CASE eState OF
    CFF_IDLE:
        bBusy := FALSE;
        bDone := FALSE;
        bError := FALSE;
        bAborted := FALSE;
        stFastConfigSnapshot.bValid := FALSE;
        IF bStartEvent THEN
            udiActiveStartCommandId := GVL_FastInternal.stAcceptedCommand.stSequence.nCommandId;
            stActiveSequenceCommand := GVL_FastInternal.stAcceptedCommand.stSequence;
            udiActiveCycleSnapshotRevision := GVL_FastInternal.stAcceptedCommand.nCycleSnapshotRevision;
            udiStartCycleSnapshotRevisionBefore := GVL_Program.stCycleSnapshot.nSnapshotRevision;
            udiStartMachineRevisionBefore := GVL_Config.stMachine.nRevision;
            udiStartForceProfileIdBefore := GVL_Config.stZForceControl.nProfileId;
            udiStartForceProfileRevisionBefore := GVL_Config.stZForceControl.nRevision;
            udiStartRAxisProfileIdBefore := GVL_Config.stRAxis.nProfileId;
            udiStartRAxisProfileRevisionBefore := GVL_Config.stRAxis.nRevision;
            stCycleSnapshot := GVL_Program.stCycleSnapshot;
            stMachineSnapshot := GVL_Config.stMachine;
            stLimitsSnapshot := GVL_Config.stLimits;
            stSequenceConfigSnapshot := GVL_Config.stCffSequence;
            stZExtConfigSnapshot := GVL_Config.stZExtSetpoint;
            stForceProfileSnapshot := GVL_Config.stZForceControl;
            stRAxisProfileSnapshot := GVL_Config.stRAxis;
            bStartSourceSnapshotConsistent :=
                (udiStartCycleSnapshotRevisionBefore = stCycleSnapshot.nSnapshotRevision)
                AND (GVL_Program.stCycleSnapshot.nSnapshotRevision
                    = stCycleSnapshot.nSnapshotRevision)
                AND (udiStartMachineRevisionBefore = stMachineSnapshot.nRevision)
                AND (GVL_Config.stMachine.nRevision = stMachineSnapshot.nRevision)
                AND (udiStartForceProfileIdBefore = stForceProfileSnapshot.nProfileId)
                AND (udiStartForceProfileRevisionBefore = stForceProfileSnapshot.nRevision)
                AND (GVL_Config.stZForceControl.nProfileId = stForceProfileSnapshot.nProfileId)
                AND (GVL_Config.stZForceControl.nRevision = stForceProfileSnapshot.nRevision)
                AND (udiStartRAxisProfileIdBefore = stRAxisProfileSnapshot.nProfileId)
                AND (udiStartRAxisProfileRevisionBefore = stRAxisProfileSnapshot.nRevision)
                AND (GVL_Config.stRAxis.nProfileId = stRAxisProfileSnapshot.nProfileId)
                AND (GVL_Config.stRAxis.nRevision = stRAxisProfileSnapshot.nRevision);
            rCycleStartZPosition_mm := GVL_Status.stFast.stZAxis.rActualPosition_mm;
            bBusy := TRUE;
            bCycleNokLatched := FALSE;
            bStopRequestedLatched := FALSE;
            bResetPendingLatched := FALSE;
            udiFirstFaultId :=0;
            eExitIntent := CFF_EXIT_NONE;
            eStep := CFF_STEP_NONE;
            eSubPhase := STEP_SUBPHASE_NONE;
            eEndCause := STEP_END_NONE;
            FOR nStepIndex := 1 TO 4 DO
                GVL_Process.astStepCriterion[nStepIndex] := stClearedStepCriterionResult;
                abStepResultWritten[nStepIndex] := FALSE;
            END_FOR
            stLastPublishedRCommand.bEnable := TRUE;
            stLastPublishedRCommand.bReset := FALSE;
            stLastPublishedRCommand.bStop := TRUE;
            stLastPublishedRCommand.bMoveVelocity := FALSE;
            stLastPublishedRCommand.rVelocity_rpm := 0.0;
            stLastPublishedRCommand.rAcceleration_rpm_s :=
                stRAxisProfileSnapshot.fSpeedRampRpmS;
            stLastPublishedRCommand.rDeceleration_rpm_s :=
                stRAxisProfileSnapshot.fSpeedRampRpmS;
            stCandidateRCommand := stLastPublishedRCommand;
            rHardMaximumRelativePosition_mm := 0.0;
            rRequiredRelativePosition_mm := 0.0;
            rStepBoundary_mm := 0.0;
            rForceTransferVelocity_mm_s := 0.0;
            rForceSet_kN := 0.0;
            rForceRamp_kN_s := 0.0;
            rSpeedSet_rpm := 0.0;
            rTargetRelativePosition_mm := 0.0;
            rStepTime_s := 0.0;
            rQualifiedForceHoldTime_s := 0.0;
            uliStepElapsed_us := 0;
            uliStepMaximum_us := 0;
            uliQualifiedHold_us := 0;
            uliQualifiedHoldTarget_us := 0;
            bRpmStopped := FALSE;
            bForceInBand := FALSE;
            bHardForceActive := FALSE;
            bHardStrokeActive := FALSE;
            bCollisionLimitActive := FALSE;
            bForceControlEnable := FALSE;
            bForceProfileTransfer := FALSE;
            bForceProfileTransferPending := FALSE;
            bProcessReferencePending := FALSE;
            bProcessReferenceResetPending := FALSE;
            bProcessReferenceLatchPending := FALSE;
            bApproachFaultStopPending := FALSE;
            bUnknownExternalRStopPending := FALSE;
            bSafeExitRStopPending := FALSE;
            bTerminalFaultStopRequired := FALSE;
            bUnloadTransferInitialized := FALSE;
            stFastConfigSnapshot.bValid := FALSE;
            eNextState := CFF_PRECHECK;
        END_IF

    CFF_PRECHECK:
        (* Generate the first of the two local Contact transactions: Reset. *)
        IF bStateEntry THEN
            IF NOT bProcessReferencePending THEN
                stPendingProcessReferenceCommand.bLatchContactReference := FALSE;
                stPendingProcessReferenceCommand.bUseProvidedContactReference := FALSE;
                stPendingProcessReferenceCommand.rProvidedContactSensorPosition_mm := 0.0;
                stPendingProcessReferenceCommand.rProvidedContactAxisPosition_mm := 0.0;
                stPendingProcessReferenceCommand.bResetContactReference := TRUE;
                udiContactReferenceRequestId := udiContactReferenceRequestId + 1;
                IF udiContactReferenceRequestId = 0 THEN
                    udiContactReferenceRequestId := 1;
                END_IF
                stPendingProcessReferenceCommand.udiContactReferenceRequestId := udiContactReferenceRequestId;
                udiExpectedContactReferenceAckId := udiContactReferenceRequestId;
                bProcessReferencePending := TRUE;
                bProcessReferenceResetPending := TRUE;
                bProcessReferenceLatchPending := FALSE;
            END_IF
        END_IF

        IF bProcessReferenceResetPending
            AND (GVL_Process.stActual.udiContactReferenceAcceptedId
                = udiExpectedContactReferenceAckId) THEN
            bProcessReferencePending := FALSE;
            bProcessReferenceResetPending := FALSE;
            IF GVL_Process.stActual.bContactReferenceValid THEN
                IF udiFirstFaultId = 0 THEN
                    udiFirstFaultId := 16#0000A001;
                END_IF
                eNextState := CFF_FAULT;
            ELSIF bPermissionValid AND bSnapshotIdentityValid
                AND stMachineSnapshot.bValid AND stLimitsSnapshot.bValid
                AND stCycleSnapshot.stProgram.bValid AND stZExtConfigSnapshot.bValid
                AND bProgramValid AND bSequenceConfigValid AND bProfileValid
                AND bHardwareReady AND bSensorReady AND bLocalReturnTargetValid
                AND bExternalReady
                AND (GVL_Status.stFast.stZAxis.eActiveOwner = Z_OWNER_NONE) THEN
                stFastConfigSnapshot.nSequenceCommandId := udiActiveStartCommandId;
                stFastConfigSnapshot.stMachine := stMachineSnapshot;
                stFastConfigSnapshot.stLimits := stLimitsSnapshot;
                stFastConfigSnapshot.stZExtSetpoint := stZExtConfigSnapshot;
                stFastConfigSnapshot.stZForceControl := stForceProfileSnapshot;
                stFastConfigSnapshot.bValid := TRUE;
                eNextState := CFF_APPROACH;
            ELSE
                IF udiFirstFaultId = 0 THEN
                    IF NOT bPermissionValid OR NOT bSnapshotIdentityValid THEN
                        udiFirstFaultId := 16#0000A001;
                    ELSIF NOT bProgramValid THEN
                        udiFirstFaultId := 16#0000A002;
                    ELSIF NOT bSequenceConfigValid OR NOT stMachineSnapshot.bValid
                        OR NOT stLimitsSnapshot.bValid OR NOT stZExtConfigSnapshot.bValid THEN
                        udiFirstFaultId := 16#0000A003;
                    ELSIF NOT bProfileValid THEN
                        udiFirstFaultId := 16#0000A004;
                    ELSIF NOT bHardwareReady THEN
                        udiFirstFaultId := 16#0000A005;
                    ELSE
                        udiFirstFaultId := 16#0000A006;
                    END_IF
                END_IF
                stFastConfigSnapshot.bValid := FALSE;
                eExitIntent := CFF_EXIT_FAULT_NO_RETURN;
                eNextState := CFF_FAULT;
            END_IF
        ELSIF tonContactReferenceAck.Q THEN
            IF udiFirstFaultId = 0 THEN
                udiFirstFaultId := 16#0000A009;
            END_IF
            stFastConfigSnapshot.bValid := FALSE;
            eExitIntent := CFF_EXIT_FAULT_NO_RETURN;
            eNextState := CFF_FAULT;
        END_IF

    CFF_APPROACH:
        stMotionIntent.stZCommand.bEnable := TRUE;
        stMotionIntent.stZCommand.bReset := FALSE;
        stMotionIntent.stZCommand.bStop := FALSE;
        stMotionIntent.stZCommand.bHome := FALSE;
        stMotionIntent.stZCommand.bMoveAbsolute := TRUE;
        stMotionIntent.stZCommand.bMoveVelocity := FALSE;
        stMotionIntent.stZCommand.bUseExternalSetpoint := FALSE;
        stMotionIntent.stZCommand.rPosition_mm := stCycleSnapshot.stProgram.stHeader.fContactSearchStartPositionMm;
        stMotionIntent.stZCommand.rVelocity_mm_s := stCycleSnapshot.stProgram.stHeader.fContactSearchVelocityMmS;
        stMotionIntent.stZCommand.rAcceleration_mm_s2 := stSequenceConfigSnapshot.fStandardMoveAccelerationMmS2;
        stMotionIntent.stZCommand.rDeceleration_mm_s2 := stSequenceConfigSnapshot.fStandardMoveDecelerationMmS2;
        stMotionIntent.stZCommand.eOwnerRequest := Z_OWNER_APPROACH;
        stMotionIntent.bRAxisProcessRequested := TRUE;
        stMotionIntent.stRCommand.bEnable := TRUE;
        stMotionIntent.stRCommand.bReset := FALSE;
        stMotionIntent.stRCommand.bStop := TRUE;
        stMotionIntent.stRCommand.bMoveVelocity := FALSE;
        stMotionIntent.stRCommand.rVelocity_rpm := 0.0;
        stMotionIntent.stRCommand.rAcceleration_rpm_s := stRAxisProfileSnapshot.fSpeedRampRpmS;
        stMotionIntent.stRCommand.rDeceleration_rpm_s := stRAxisProfileSnapshot.fSpeedRampRpmS;
        IF bStateEntry THEN
            IF bEntryMotionPermitted THEN
                udiZCommandId := udiZCommandId + 1;
                IF udiZCommandId = 0 THEN
                    udiZCommandId := 1;
                END_IF
            END_IF
            udiRCommandId := udiRCommandId + 1;
            IF udiRCommandId = 0 THEN
                udiRCommandId := 1;
            END_IF
        END_IF
        IF bApproachNormalCompletion THEN
            eNextState := CFF_EXTSETPOINT_PREPARE;
        ELSIF tonRAxisStop.Q THEN
            IF udiFirstFaultId = 0 THEN
                udiFirstFaultId := 16#0000A014;
            END_IF
            eExitIntent := CFF_EXIT_FAULT_NO_RETURN;
            eNextState := CFF_FAULT;
        ELSIF tonApproach.Q THEN
            IF udiFirstFaultId = 0 THEN
                udiFirstFaultId := 16#0000A007;
            END_IF
            eExitIntent := CFF_EXIT_FAULT_NO_RETURN;
            eNextState := CFF_FAULT;
        ELSIF GVL_Status.stFast.stZAxis.bError THEN
            IF udiFirstFaultId = 0 THEN
                udiFirstFaultId := 16#0000A010;
            END_IF
            eExitIntent := CFF_EXIT_FAULT_NO_RETURN;
            eNextState := CFF_FAULT;
        ELSIF GVL_Status.stFast.stRAxis.bError THEN
            IF udiFirstFaultId = 0 THEN
                udiFirstFaultId := 16#0000A011;
            END_IF
            eExitIntent := CFF_EXIT_FAULT_NO_RETURN;
            eNextState := CFF_FAULT;
        END_IF

    CFF_EXTSETPOINT_PREPARE:
        stMotionIntent.stZCommand.bEnable := TRUE;
        stMotionIntent.stZCommand.bUseExternalSetpoint := TRUE;
        stMotionIntent.stZCommand.eOwnerRequest := Z_OWNER_FORCE_PROCESS;
        stMotionIntent.bExternalEnableRequest := TRUE;
        stMotionIntent.bExternalDisableRequest := FALSE;
        stMotionIntent.bRAxisProcessRequested := TRUE;
        stMotionIntent.stRCommand.bEnable := TRUE;
        stMotionIntent.stRCommand.bStop := TRUE;
        stMotionIntent.stRCommand.bMoveVelocity := FALSE;
        stMotionIntent.stRCommand.rVelocity_rpm := 0.0;
        stMotionIntent.stRCommand.rAcceleration_rpm_s := stRAxisProfileSnapshot.fSpeedRampRpmS;
        stMotionIntent.stRCommand.rDeceleration_rpm_s := stRAxisProfileSnapshot.fSpeedRampRpmS;
        bForceControlEnable := FALSE;
        IF bStateEntry THEN
            udiZCommandId := udiZCommandId + 1;
            IF udiZCommandId = 0 THEN
                udiZCommandId := 1;
            END_IF
        END_IF
        IF (GVL_Status.stFast.udiAcceptedSequenceZCommandId = udiZCommandId)
            AND (GVL_Status.stFast.stZAxis.eActiveOwner = Z_OWNER_FORCE_PROCESS)
            AND GVL_Status.stFast.stZExtSetpoint.bEnabled
            AND GVL_Status.stFast.stZExtSetpoint.bAcceptedSetpointValid
            AND GVL_Status.stFast.stZExternalTrajectory.bActive THEN
            eNextState := CFF_CONTACT_SEARCH;
        END_IF

    CFF_CONTACT_SEARCH:
        stMotionIntent.stZCommand.bEnable := TRUE;
        stMotionIntent.stZCommand.bUseExternalSetpoint := TRUE;
        stMotionIntent.stZCommand.eOwnerRequest := Z_OWNER_FORCE_PROCESS;
        stMotionIntent.bExternalEnableRequest := TRUE;
        stMotionIntent.bExternalDisableRequest := FALSE;
        stMotionIntent.rExternalTargetVelocity_mm_s := ABS(stCycleSnapshot.stProgram.stHeader.fContactSearchVelocityMmS);
        stMotionIntent.bRAxisProcessRequested := TRUE;
        stMotionIntent.stRCommand.bEnable := TRUE;
        stMotionIntent.stRCommand.bStop := TRUE;
        stMotionIntent.stRCommand.bMoveVelocity := FALSE;
        stMotionIntent.stRCommand.rVelocity_rpm := 0.0;
        stMotionIntent.stRCommand.rAcceleration_rpm_s := stRAxisProfileSnapshot.fSpeedRampRpmS;
        stMotionIntent.stRCommand.rDeceleration_rpm_s := stRAxisProfileSnapshot.fSpeedRampRpmS;
        bForceControlEnable := FALSE;
        IF fbContactDetect.stOutput.bReferenceLatchRequest AND NOT bProcessReferencePending THEN
            stPendingProcessReferenceCommand.bLatchContactReference := TRUE;
            stPendingProcessReferenceCommand.bUseProvidedContactReference := TRUE;
            stPendingProcessReferenceCommand.rProvidedContactSensorPosition_mm := fbContactDetect.stOutput.rDetectedSensorPosition_mm;
            stPendingProcessReferenceCommand.rProvidedContactAxisPosition_mm := fbContactDetect.stOutput.rDetectedAxisPosition_mm;
            stPendingProcessReferenceCommand.bResetContactReference := FALSE;
            udiContactReferenceRequestId := udiContactReferenceRequestId + 1;
            IF udiContactReferenceRequestId = 0 THEN
                udiContactReferenceRequestId := 1;
            END_IF
            stPendingProcessReferenceCommand.udiContactReferenceRequestId := udiContactReferenceRequestId;
            udiExpectedContactReferenceAckId := udiContactReferenceRequestId;
            bProcessReferencePending := TRUE;
            bProcessReferenceResetPending := FALSE;
            bProcessReferenceLatchPending := TRUE;
            eNextState := CFF_CONTACT_ACCEPT;
        ELSIF tonContactSearch.Q OR fbContactDetect.stOutput.bFault THEN
            IF udiFirstFaultId = 0 THEN
                udiFirstFaultId := 16#0000A008;
            END_IF
            eExitIntent := CFF_EXIT_FAULT_NO_RETURN;
            eNextState := CFF_EXTSETPOINT_DISABLE;
        END_IF

    CFF_CONTACT_ACCEPT:
        stMotionIntent.stZCommand.bEnable := TRUE;
        stMotionIntent.stZCommand.bUseExternalSetpoint := TRUE;
        stMotionIntent.stZCommand.eOwnerRequest := Z_OWNER_FORCE_PROCESS;
        stMotionIntent.bExternalEnableRequest := TRUE;
        stMotionIntent.bExternalDisableRequest := FALSE;
        stMotionIntent.rExternalTargetVelocity_mm_s := ABS(stCycleSnapshot.stProgram.stHeader.fContactSearchVelocityMmS);
        stMotionIntent.bRAxisProcessRequested := TRUE;
        stMotionIntent.stRCommand.bEnable := TRUE;
        stMotionIntent.stRCommand.bStop := TRUE;
        stMotionIntent.stRCommand.bMoveVelocity := FALSE;
        stMotionIntent.stRCommand.rVelocity_rpm := 0.0;
        stMotionIntent.stRCommand.rAcceleration_rpm_s := stRAxisProfileSnapshot.fSpeedRampRpmS;
        stMotionIntent.stRCommand.rDeceleration_rpm_s := stRAxisProfileSnapshot.fSpeedRampRpmS;
        bForceControlEnable := FALSE;
        IF bProcessReferenceLatchPending
            AND (GVL_Process.stActual.udiContactReferenceAcceptedId
                = udiExpectedContactReferenceAckId) THEN
            bProcessReferencePending := FALSE;
            bProcessReferenceLatchPending := FALSE;
            IF NOT GVL_Process.stActual.bContactReferenceValid THEN
                IF udiFirstFaultId = 0 THEN
                    udiFirstFaultId := 16#0000A00A;
                END_IF
                eExitIntent := CFF_EXIT_FAULT_NO_RETURN;
                eNextState := CFF_EXTSETPOINT_DISABLE;
            ELSIF NOT GVL_Process.stActual.bAxisSensorAgreement
                OR NOT GVL_Process.stActual.bValid THEN
                IF udiFirstFaultId = 0 THEN
                    udiFirstFaultId := 16#0000A00F;
                END_IF
                eExitIntent := CFF_EXIT_FAULT_NO_RETURN;
                eNextState := CFF_EXTSETPOINT_DISABLE;
            ELSE
                rHardMaximumRelativePosition_mm := stLimitsSnapshot.fZMaxPositionMm
                    - GVL_Process.stActual.fContactAxisPositionMm;
                rRequiredRelativePosition_mm := 0.0;
                FOR nStepIndex := 1 TO 4 DO
                    rStepBoundary_mm := stCycleSnapshot.stProgram.astSteps[nStepIndex].stProceeding.fRelativeDistanceMm;
                    IF stCycleSnapshot.stProgram.astSteps[nStepIndex].stProceeding.fSecondarySRelMm
                        > rStepBoundary_mm THEN
                        rStepBoundary_mm := stCycleSnapshot.stProgram.astSteps[nStepIndex].stProceeding.fSecondarySRelMm;
                    END_IF
                    IF rStepBoundary_mm > rRequiredRelativePosition_mm THEN
                        rRequiredRelativePosition_mm := rStepBoundary_mm;
                    END_IF
                END_FOR
                IF NOT FC_IsFiniteLReal(rValue := rHardMaximumRelativePosition_mm)
                    OR (rHardMaximumRelativePosition_mm <= 0.0)
                    OR (rRequiredRelativePosition_mm > rHardMaximumRelativePosition_mm) THEN
                    IF udiFirstFaultId = 0 THEN
                        udiFirstFaultId := 16#0000A00D;
                    END_IF
                    eExitIntent := CFF_EXIT_FAULT_NO_RETURN;
                    eNextState := CFF_EXTSETPOINT_DISABLE;
                ELSE
                    rForceTransferVelocity_mm_s := GVL_Status.stFast.stZExtSetpoint.rAcceptedVelocity_mm_s;
                    rForceSet_kN := GVL_Process.stActual.fForceControlN * 0.001;
                    rForceRamp_kN_s := stForceProfileSnapshot.fForceRampNS * 0.001;
                    bForceProfileTransferPending := TRUE;
                    bForceControlEnable := TRUE;
                    eNextState := CFF_STEP1_ENTRY;
                END_IF
            END_IF
        ELSIF tonContactReferenceAck.Q THEN
            IF udiFirstFaultId = 0 THEN
                udiFirstFaultId := 16#0000A009;
            END_IF
            eExitIntent := CFF_EXIT_FAULT_NO_RETURN;
            eNextState := CFF_EXTSETPOINT_DISABLE;
        END_IF

    (* Step1 Entry：同一扫描发布Force目标、R目标和一次事务。 *)
    CFF_STEP1_ENTRY:
        stMotionIntent.stZCommand.bEnable := TRUE;
        stMotionIntent.stZCommand.bUseExternalSetpoint := TRUE;
        stMotionIntent.stZCommand.eOwnerRequest := Z_OWNER_FORCE_PROCESS;
        stMotionIntent.bExternalEnableRequest := TRUE;
        stMotionIntent.bRAxisProcessRequested := TRUE;
        stMotionIntent.stRCommand := stLastPublishedRCommand;
        bForceControlEnable := TRUE;
        eStep := CFF_STEP1_PENETRATION;
        eSubPhase := STEP_SUBPHASE_ENTRY;
        IF bStateEntry AND bEntryMotionPermitted THEN
            rForceSet_kN := stCycleSnapshot.stProgram.astSteps[1].fSetForceN * 0.001;
            rForceRamp_kN_s := stCycleSnapshot.stProgram.astSteps[1].fForceRampNS * 0.001;
            rSpeedSet_rpm := stCycleSnapshot.stProgram.astSteps[1].fSetSpeedRpm;
            IF stCycleSnapshot.stProgram.astSteps[nActiveStepProgramIndex].stProceeding.ePrimaryCriterion
                = STEP_CRIT_RELATIVE_DISTANCE THEN
                rTargetRelativePosition_mm :=
                    stCycleSnapshot.stProgram.astSteps[nActiveStepProgramIndex].stProceeding.fRelativeDistanceMm;
            ELSE
                rTargetRelativePosition_mm :=
                    stCycleSnapshot.stProgram.astSteps[nActiveStepProgramIndex].stProceeding.fSecondarySRelMm;
            END_IF
            rForceTransferVelocity_mm_s :=
                GVL_Status.stFast.stZExtSetpoint.rAcceptedVelocity_mm_s;
            bForceProfileTransferPending := TRUE;
            stMotionIntent.stRCommand := stCandidateRCommand;
            IF bRCommandPayloadChanged THEN
                stLastPublishedRCommand := stCandidateRCommand;
                stMotionIntent.stRCommand := stCandidateRCommand;
                udiRCommandId := udiRCommandId + 1;
                IF udiRCommandId = 0 THEN
                    udiRCommandId := 1;
                END_IF
            END_IF
            eNextState := CFF_STEP1_RAMP_PROCESS;
        END_IF

    (* Step1 Process：每扫描完整执行Decline与Criterion。 *)
    CFF_STEP1_RAMP_PROCESS:
        stMotionIntent.stZCommand.bEnable := TRUE;
        stMotionIntent.stZCommand.bUseExternalSetpoint := TRUE;
        stMotionIntent.stZCommand.eOwnerRequest := Z_OWNER_FORCE_PROCESS;
        stMotionIntent.bExternalEnableRequest := TRUE;
        stMotionIntent.bRAxisProcessRequested := TRUE;
        stMotionIntent.stRCommand := stLastPublishedRCommand;
        bForceControlEnable := TRUE;
        eStep := CFF_STEP1_PENETRATION;
        eSubPhase := STEP_SUBPHASE_RAMP_PROCESS;
        IF udiFirstFaultId > 0 THEN
            IF fbStepCriterion.stOutput.bEndConfirmed
                AND ((fbStepCriterion.stOutput.eEndCause = STEP_END_HARD_FORCE)
                    OR (fbStepCriterion.stOutput.eEndCause = STEP_END_HARD_STROKE)
                    OR (fbStepCriterion.stOutput.eEndCause = STEP_END_COLLISION)
                    OR (fbStepCriterion.stOutput.eEndCause = STEP_END_SENSOR_INVALID)
                    OR (fbStepCriterion.stOutput.eEndCause = STEP_END_AXIS_FAULT))
                AND NOT fbForceDecline.stOutput.bFault
                AND NOT fbStepCriterion.stOutput.bFault THEN
                nStepResultIndex := 1;
                bStepResultNok := TRUE;
                bStepResultPublishRequested := TRUE;
                eEndCause := fbStepCriterion.stOutput.eEndCause;
            END_IF
            eExitIntent := CFF_EXIT_FAULT_NO_RETURN;
            eNextState := CFF_EXTSETPOINT_DISABLE;
        ELSIF fbForceDecline.stOutput.bFault OR fbStepCriterion.stOutput.bFault THEN
            IF udiFirstFaultId = 0 THEN
                udiFirstFaultId := 16#0000A00B;
            END_IF
            eExitIntent := CFF_EXIT_FAULT_NO_RETURN;
            eNextState := CFF_EXTSETPOINT_DISABLE;
        ELSIF fbStepCriterion.stOutput.bEndConfirmed THEN
            nStepResultIndex := 1;
            bStepResultNok := fbStepCriterion.stOutput.bNok;
            bStepResultPublishRequested := TRUE;
            eEndCause := fbStepCriterion.stOutput.eEndCause;
            IF udiFirstFaultId > 0 THEN
                eExitIntent := CFF_EXIT_FAULT_NO_RETURN;
                eNextState := CFF_EXTSETPOINT_DISABLE;
            ELSIF bStopRequestedLatched OR bAbortEvent OR bResetPendingLatched THEN
                eExitIntent := CFF_EXIT_ABORT_NO_RETURN;
                eNextState := CFF_EXTSETPOINT_DISABLE;
            ELSE
                eNextState := CFF_STEP1_END_CHECK;
            END_IF
        END_IF

    (* Step1 End：只锁存一次真实结果，然后推进或受控卸载。 *)
    CFF_STEP1_END_CHECK:
        stMotionIntent.stZCommand.bEnable := TRUE;
        stMotionIntent.stZCommand.bUseExternalSetpoint := TRUE;
        stMotionIntent.stZCommand.eOwnerRequest := Z_OWNER_FORCE_PROCESS;
        stMotionIntent.bExternalEnableRequest := TRUE;
        stMotionIntent.bRAxisProcessRequested := TRUE;
        stMotionIntent.stRCommand := stLastPublishedRCommand;
        bForceControlEnable := TRUE;
        eStep := CFF_STEP1_PENETRATION;
        eSubPhase := STEP_SUBPHASE_END_CHECK;
        IF udiFirstFaultId > 0 THEN
            eExitIntent := CFF_EXIT_FAULT_NO_RETURN;
            eNextState := CFF_EXTSETPOINT_DISABLE;
        ELSIF bStopRequestedLatched OR bAbortEvent OR bResetPendingLatched THEN
            IF fbStepCriterion.stOutput.bEndConfirmed
                AND (fbStepCriterion.stOutput.eEndCause = STEP_END_STOP_REQUEST)
                AND NOT fbForceDecline.stOutput.bFault
                AND NOT fbStepCriterion.stOutput.bFault THEN
                nStepResultIndex := 1;
                bStepResultNok := fbStepCriterion.stOutput.bNok;
                bStepResultPublishRequested := TRUE;
                eEndCause := fbStepCriterion.stOutput.eEndCause;
            END_IF
            eExitIntent := CFF_EXIT_ABORT_NO_RETURN;
            eNextState := CFF_EXTSETPOINT_DISABLE;
        ELSIF fbForceDecline.stOutput.bFault OR fbStepCriterion.stOutput.bFault THEN
            IF udiFirstFaultId = 0 THEN
                udiFirstFaultId := 16#0000A00B;
            END_IF
            eExitIntent := CFF_EXIT_FAULT_NO_RETURN;
            eNextState := CFF_EXTSETPOINT_DISABLE;
        ELSIF fbStepCriterion.stOutput.bEndConfirmed THEN
            nStepResultIndex := 1;
            bStepResultNok := fbStepCriterion.stOutput.bNok;
            bStepResultPublishRequested := TRUE;
            eEndCause := fbStepCriterion.stOutput.eEndCause;
            IF fbStepCriterion.stOutput.bNok THEN
                bCycleNokLatched := TRUE;
            END_IF
            IF fbStepCriterion.stOutput.bControlledExitRequested
                AND NOT fbStepCriterion.stOutput.bAdvanceRequested THEN
                eExitIntent := CFF_EXIT_NOK_RETURN;
                eNextState := CFF_CONTROLLED_FORCE_UNLOAD;
            ELSIF fbStepCriterion.stOutput.bAdvanceRequested THEN
                eNextState := CFF_STEP2_ENTRY;
            ELSE
                IF udiFirstFaultId = 0 THEN
                    udiFirstFaultId := 16#0000A00B;
                END_IF
                eExitIntent := CFF_EXIT_FAULT_NO_RETURN;
                eNextState := CFF_EXTSETPOINT_DISABLE;
            END_IF
        END_IF

    (* Step2 Entry：Force Profile更新与R完整payload去重。 *)
    CFF_STEP2_ENTRY:
        stMotionIntent.stZCommand.bEnable := TRUE;
        stMotionIntent.stZCommand.bUseExternalSetpoint := TRUE;
        stMotionIntent.stZCommand.eOwnerRequest := Z_OWNER_FORCE_PROCESS;
        stMotionIntent.bExternalEnableRequest := TRUE;
        stMotionIntent.bRAxisProcessRequested := TRUE;
        stMotionIntent.stRCommand := stLastPublishedRCommand;
        bForceControlEnable := TRUE;
        eStep := CFF_STEP2_CLEAN_ACTIVATE;
        eSubPhase := STEP_SUBPHASE_ENTRY;
        IF bStateEntry AND bEntryMotionPermitted THEN
            rForceSet_kN := stCycleSnapshot.stProgram.astSteps[2].fSetForceN * 0.001;
            rForceRamp_kN_s := stCycleSnapshot.stProgram.astSteps[2].fForceRampNS * 0.001;
            rSpeedSet_rpm := stCycleSnapshot.stProgram.astSteps[2].fSetSpeedRpm;
            IF stCycleSnapshot.stProgram.astSteps[nActiveStepProgramIndex].stProceeding.ePrimaryCriterion
                = STEP_CRIT_RELATIVE_DISTANCE THEN
                rTargetRelativePosition_mm :=
                    stCycleSnapshot.stProgram.astSteps[nActiveStepProgramIndex].stProceeding.fRelativeDistanceMm;
            ELSE
                rTargetRelativePosition_mm :=
                    stCycleSnapshot.stProgram.astSteps[nActiveStepProgramIndex].stProceeding.fSecondarySRelMm;
            END_IF
            rForceTransferVelocity_mm_s :=
                GVL_Status.stFast.stZExtSetpoint.rAcceptedVelocity_mm_s;
            bForceProfileTransferPending := TRUE;
            stMotionIntent.stRCommand := stCandidateRCommand;
            IF bRCommandPayloadChanged THEN
                stLastPublishedRCommand := stCandidateRCommand;
                stMotionIntent.stRCommand := stCandidateRCommand;
                udiRCommandId := udiRCommandId + 1;
                IF udiRCommandId = 0 THEN
                    udiRCommandId := 1;
                END_IF
            END_IF
            eNextState := CFF_STEP2_RAMP_PROCESS;
        END_IF

    CFF_STEP2_RAMP_PROCESS:
        stMotionIntent.stZCommand.bEnable := TRUE;
        stMotionIntent.stZCommand.bUseExternalSetpoint := TRUE;
        stMotionIntent.stZCommand.eOwnerRequest := Z_OWNER_FORCE_PROCESS;
        stMotionIntent.bExternalEnableRequest := TRUE;
        stMotionIntent.bRAxisProcessRequested := TRUE;
        stMotionIntent.stRCommand := stLastPublishedRCommand;
        bForceControlEnable := TRUE;
        eStep := CFF_STEP2_CLEAN_ACTIVATE;
        eSubPhase := STEP_SUBPHASE_RAMP_PROCESS;
        IF udiFirstFaultId > 0 THEN
            IF fbStepCriterion.stOutput.bEndConfirmed
                AND ((fbStepCriterion.stOutput.eEndCause = STEP_END_HARD_FORCE)
                    OR (fbStepCriterion.stOutput.eEndCause = STEP_END_HARD_STROKE)
                    OR (fbStepCriterion.stOutput.eEndCause = STEP_END_COLLISION)
                    OR (fbStepCriterion.stOutput.eEndCause = STEP_END_SENSOR_INVALID)
                    OR (fbStepCriterion.stOutput.eEndCause = STEP_END_AXIS_FAULT))
                AND NOT fbForceDecline.stOutput.bFault
                AND NOT fbStepCriterion.stOutput.bFault THEN
                nStepResultIndex := 2;
                bStepResultNok := TRUE;
                bStepResultPublishRequested := TRUE;
                eEndCause := fbStepCriterion.stOutput.eEndCause;
            END_IF
            eExitIntent := CFF_EXIT_FAULT_NO_RETURN;
            eNextState := CFF_EXTSETPOINT_DISABLE;
        ELSIF fbForceDecline.stOutput.bFault OR fbStepCriterion.stOutput.bFault THEN
            IF udiFirstFaultId = 0 THEN
                udiFirstFaultId := 16#0000A00B;
            END_IF
            eExitIntent := CFF_EXIT_FAULT_NO_RETURN;
            eNextState := CFF_EXTSETPOINT_DISABLE;
        ELSIF fbStepCriterion.stOutput.bEndConfirmed THEN
            nStepResultIndex := 2;
            bStepResultNok := fbStepCriterion.stOutput.bNok;
            bStepResultPublishRequested := TRUE;
            eEndCause := fbStepCriterion.stOutput.eEndCause;
            IF udiFirstFaultId > 0 THEN
                eExitIntent := CFF_EXIT_FAULT_NO_RETURN;
                eNextState := CFF_EXTSETPOINT_DISABLE;
            ELSIF bStopRequestedLatched OR bAbortEvent OR bResetPendingLatched THEN
                eExitIntent := CFF_EXIT_ABORT_NO_RETURN;
                eNextState := CFF_EXTSETPOINT_DISABLE;
            ELSE
                eNextState := CFF_STEP2_END_CHECK;
            END_IF
        END_IF

    CFF_STEP2_END_CHECK:
        stMotionIntent.stZCommand.bEnable := TRUE;
        stMotionIntent.stZCommand.bUseExternalSetpoint := TRUE;
        stMotionIntent.stZCommand.eOwnerRequest := Z_OWNER_FORCE_PROCESS;
        stMotionIntent.bExternalEnableRequest := TRUE;
        stMotionIntent.bRAxisProcessRequested := TRUE;
        stMotionIntent.stRCommand := stLastPublishedRCommand;
        bForceControlEnable := TRUE;
        eStep := CFF_STEP2_CLEAN_ACTIVATE;
        eSubPhase := STEP_SUBPHASE_END_CHECK;
        IF udiFirstFaultId > 0 THEN
            eExitIntent := CFF_EXIT_FAULT_NO_RETURN;
            eNextState := CFF_EXTSETPOINT_DISABLE;
        ELSIF bStopRequestedLatched OR bAbortEvent OR bResetPendingLatched THEN
            IF fbStepCriterion.stOutput.bEndConfirmed
                AND (fbStepCriterion.stOutput.eEndCause = STEP_END_STOP_REQUEST)
                AND NOT fbForceDecline.stOutput.bFault
                AND NOT fbStepCriterion.stOutput.bFault THEN
                nStepResultIndex := 2;
                bStepResultNok := fbStepCriterion.stOutput.bNok;
                bStepResultPublishRequested := TRUE;
                eEndCause := fbStepCriterion.stOutput.eEndCause;
            END_IF
            eExitIntent := CFF_EXIT_ABORT_NO_RETURN;
            eNextState := CFF_EXTSETPOINT_DISABLE;
        ELSIF fbForceDecline.stOutput.bFault OR fbStepCriterion.stOutput.bFault THEN
            IF udiFirstFaultId = 0 THEN
                udiFirstFaultId := 16#0000A00B;
            END_IF
            eExitIntent := CFF_EXIT_FAULT_NO_RETURN;
            eNextState := CFF_EXTSETPOINT_DISABLE;
        ELSIF fbStepCriterion.stOutput.bEndConfirmed THEN
            nStepResultIndex := 2;
            bStepResultNok := fbStepCriterion.stOutput.bNok;
            bStepResultPublishRequested := TRUE;
            eEndCause := fbStepCriterion.stOutput.eEndCause;
            IF fbStepCriterion.stOutput.bNok THEN
                bCycleNokLatched := TRUE;
            END_IF
            IF fbStepCriterion.stOutput.bControlledExitRequested
                AND NOT fbStepCriterion.stOutput.bAdvanceRequested THEN
                eExitIntent := CFF_EXIT_NOK_RETURN;
                eNextState := CFF_CONTROLLED_FORCE_UNLOAD;
            ELSIF fbStepCriterion.stOutput.bAdvanceRequested THEN
                eNextState := CFF_STEP3_ENTRY;
            ELSE
                IF udiFirstFaultId = 0 THEN
                    udiFirstFaultId := 16#0000A00B;
                END_IF
                eExitIntent := CFF_EXIT_FAULT_NO_RETURN;
                eNextState := CFF_EXTSETPOINT_DISABLE;
            END_IF
        END_IF

    (* Step3 Entry/Process/End保持同一套事务和结果合同。 *)
    CFF_STEP3_ENTRY:
        stMotionIntent.stZCommand.bEnable := TRUE;
        stMotionIntent.stZCommand.bUseExternalSetpoint := TRUE;
        stMotionIntent.stZCommand.eOwnerRequest := Z_OWNER_FORCE_PROCESS;
        stMotionIntent.bExternalEnableRequest := TRUE;
        stMotionIntent.bRAxisProcessRequested := TRUE;
        stMotionIntent.stRCommand := stLastPublishedRCommand;
        bForceControlEnable := TRUE;
        eStep := CFF_STEP3_WELDING;
        eSubPhase := STEP_SUBPHASE_ENTRY;
        IF bStateEntry AND bEntryMotionPermitted THEN
            rForceSet_kN := stCycleSnapshot.stProgram.astSteps[3].fSetForceN * 0.001;
            rForceRamp_kN_s := stCycleSnapshot.stProgram.astSteps[3].fForceRampNS * 0.001;
            rSpeedSet_rpm := stCycleSnapshot.stProgram.astSteps[3].fSetSpeedRpm;
            IF stCycleSnapshot.stProgram.astSteps[nActiveStepProgramIndex].stProceeding.ePrimaryCriterion
                = STEP_CRIT_RELATIVE_DISTANCE THEN
                rTargetRelativePosition_mm :=
                    stCycleSnapshot.stProgram.astSteps[nActiveStepProgramIndex].stProceeding.fRelativeDistanceMm;
            ELSE
                rTargetRelativePosition_mm :=
                    stCycleSnapshot.stProgram.astSteps[nActiveStepProgramIndex].stProceeding.fSecondarySRelMm;
            END_IF
            rForceTransferVelocity_mm_s :=
                GVL_Status.stFast.stZExtSetpoint.rAcceptedVelocity_mm_s;
            bForceProfileTransferPending := TRUE;
            stMotionIntent.stRCommand := stCandidateRCommand;
            IF bRCommandPayloadChanged THEN
                stLastPublishedRCommand := stCandidateRCommand;
                stMotionIntent.stRCommand := stCandidateRCommand;
                udiRCommandId := udiRCommandId + 1;
                IF udiRCommandId = 0 THEN
                    udiRCommandId := 1;
                END_IF
            END_IF
            eNextState := CFF_STEP3_RAMP_PROCESS;
        END_IF

    CFF_STEP3_RAMP_PROCESS:
        stMotionIntent.stZCommand.bEnable := TRUE;
        stMotionIntent.stZCommand.bUseExternalSetpoint := TRUE;
        stMotionIntent.stZCommand.eOwnerRequest := Z_OWNER_FORCE_PROCESS;
        stMotionIntent.bExternalEnableRequest := TRUE;
        stMotionIntent.bRAxisProcessRequested := TRUE;
        stMotionIntent.stRCommand := stLastPublishedRCommand;
        bForceControlEnable := TRUE;
        eStep := CFF_STEP3_WELDING;
        eSubPhase := STEP_SUBPHASE_RAMP_PROCESS;
        IF udiFirstFaultId > 0 THEN
            IF fbStepCriterion.stOutput.bEndConfirmed
                AND ((fbStepCriterion.stOutput.eEndCause = STEP_END_HARD_FORCE)
                    OR (fbStepCriterion.stOutput.eEndCause = STEP_END_HARD_STROKE)
                    OR (fbStepCriterion.stOutput.eEndCause = STEP_END_COLLISION)
                    OR (fbStepCriterion.stOutput.eEndCause = STEP_END_SENSOR_INVALID)
                    OR (fbStepCriterion.stOutput.eEndCause = STEP_END_AXIS_FAULT))
                AND NOT fbForceDecline.stOutput.bFault
                AND NOT fbStepCriterion.stOutput.bFault THEN
                nStepResultIndex := 3;
                bStepResultNok := TRUE;
                bStepResultPublishRequested := TRUE;
                eEndCause := fbStepCriterion.stOutput.eEndCause;
            END_IF
            eExitIntent := CFF_EXIT_FAULT_NO_RETURN;
            eNextState := CFF_EXTSETPOINT_DISABLE;
        ELSIF fbForceDecline.stOutput.bFault OR fbStepCriterion.stOutput.bFault THEN
            IF udiFirstFaultId = 0 THEN
                udiFirstFaultId := 16#0000A00B;
            END_IF
            eExitIntent := CFF_EXIT_FAULT_NO_RETURN;
            eNextState := CFF_EXTSETPOINT_DISABLE;
        ELSIF fbStepCriterion.stOutput.bEndConfirmed THEN
            nStepResultIndex := 3;
            bStepResultNok := fbStepCriterion.stOutput.bNok;
            bStepResultPublishRequested := TRUE;
            eEndCause := fbStepCriterion.stOutput.eEndCause;
            IF udiFirstFaultId > 0 THEN
                eExitIntent := CFF_EXIT_FAULT_NO_RETURN;
                eNextState := CFF_EXTSETPOINT_DISABLE;
            ELSIF bStopRequestedLatched OR bAbortEvent OR bResetPendingLatched THEN
                eExitIntent := CFF_EXIT_ABORT_NO_RETURN;
                eNextState := CFF_EXTSETPOINT_DISABLE;
            ELSE
                eNextState := CFF_STEP3_END_CHECK;
            END_IF
        END_IF

    CFF_STEP3_END_CHECK:
        stMotionIntent.stZCommand.bEnable := TRUE;
        stMotionIntent.stZCommand.bUseExternalSetpoint := TRUE;
        stMotionIntent.stZCommand.eOwnerRequest := Z_OWNER_FORCE_PROCESS;
        stMotionIntent.bExternalEnableRequest := TRUE;
        stMotionIntent.bRAxisProcessRequested := TRUE;
        stMotionIntent.stRCommand := stLastPublishedRCommand;
        bForceControlEnable := TRUE;
        eStep := CFF_STEP3_WELDING;
        eSubPhase := STEP_SUBPHASE_END_CHECK;
        IF udiFirstFaultId > 0 THEN
            eExitIntent := CFF_EXIT_FAULT_NO_RETURN;
            eNextState := CFF_EXTSETPOINT_DISABLE;
        ELSIF bStopRequestedLatched OR bAbortEvent OR bResetPendingLatched THEN
            IF fbStepCriterion.stOutput.bEndConfirmed
                AND (fbStepCriterion.stOutput.eEndCause = STEP_END_STOP_REQUEST)
                AND NOT fbForceDecline.stOutput.bFault
                AND NOT fbStepCriterion.stOutput.bFault THEN
                nStepResultIndex := 3;
                bStepResultNok := fbStepCriterion.stOutput.bNok;
                bStepResultPublishRequested := TRUE;
                eEndCause := fbStepCriterion.stOutput.eEndCause;
            END_IF
            eExitIntent := CFF_EXIT_ABORT_NO_RETURN;
            eNextState := CFF_EXTSETPOINT_DISABLE;
        ELSIF fbForceDecline.stOutput.bFault OR fbStepCriterion.stOutput.bFault THEN
            IF udiFirstFaultId = 0 THEN
                udiFirstFaultId := 16#0000A00B;
            END_IF
            eExitIntent := CFF_EXIT_FAULT_NO_RETURN;
            eNextState := CFF_EXTSETPOINT_DISABLE;
        ELSIF fbStepCriterion.stOutput.bEndConfirmed THEN
            nStepResultIndex := 3;
            bStepResultNok := fbStepCriterion.stOutput.bNok;
            bStepResultPublishRequested := TRUE;
            eEndCause := fbStepCriterion.stOutput.eEndCause;
            IF fbStepCriterion.stOutput.bNok THEN
                bCycleNokLatched := TRUE;
            END_IF
            IF fbStepCriterion.stOutput.bControlledExitRequested
                AND NOT fbStepCriterion.stOutput.bAdvanceRequested THEN
                eExitIntent := CFF_EXIT_NOK_RETURN;
                eNextState := CFF_CONTROLLED_FORCE_UNLOAD;
            ELSIF fbStepCriterion.stOutput.bAdvanceRequested THEN
                eNextState := CFF_BRAKE_AND_COMPRESSION_RAMP;
            ELSE
                IF udiFirstFaultId = 0 THEN
                    udiFirstFaultId := 16#0000A00B;
                END_IF
                eExitIntent := CFF_EXIT_FAULT_NO_RETURN;
                eNextState := CFF_EXTSETPOINT_DISABLE;
            END_IF
        END_IF

    (* Brake Entry：R停止与Step4 Force/Ramp/计时同一扫描启动。 *)
    CFF_BRAKE_AND_COMPRESSION_RAMP:
        stMotionIntent.stZCommand.bEnable := TRUE;
        stMotionIntent.stZCommand.bUseExternalSetpoint := TRUE;
        stMotionIntent.stZCommand.eOwnerRequest := Z_OWNER_FORCE_PROCESS;
        stMotionIntent.bExternalEnableRequest := TRUE;
        stMotionIntent.bRAxisProcessRequested := TRUE;
        stMotionIntent.stRCommand := stLastPublishedRCommand;
        bForceControlEnable := TRUE;
        eStep := CFF_STEP4_COMPRESSION;
        eSubPhase := STEP_SUBPHASE_BRAKE_COMPRESSION;
        IF bStateEntry AND bEntryMotionPermitted THEN
            rForceSet_kN := stCycleSnapshot.stProgram.astSteps[4].fSetForceN * 0.001;
            rForceRamp_kN_s := stCycleSnapshot.stProgram.astSteps[4].fForceRampNS * 0.001;
            rSpeedSet_rpm := 0.0;
            rTargetRelativePosition_mm :=
                stCycleSnapshot.stProgram.astSteps[4].stProceeding.fSecondarySRelMm;
            rForceTransferVelocity_mm_s :=
                GVL_Status.stFast.stZExtSetpoint.rAcceptedVelocity_mm_s;
            bForceProfileTransferPending := TRUE;
            stCandidateRCommand.rVelocity_rpm := 0.0;
            stCandidateRCommand.bEnable := TRUE;
            stCandidateRCommand.bReset := FALSE;
            stCandidateRCommand.bStop := TRUE;
            stCandidateRCommand.bMoveVelocity := FALSE;
            stCandidateRCommand.rAcceleration_rpm_s := stRAxisProfileSnapshot.fSpeedRampRpmS;
            stCandidateRCommand.rDeceleration_rpm_s := stRAxisProfileSnapshot.fSpeedRampRpmS;
            stMotionIntent.stRCommand := stCandidateRCommand;
            IF bRCommandPayloadChanged THEN
                stLastPublishedRCommand := stCandidateRCommand;
                stMotionIntent.stRCommand := stCandidateRCommand;
                udiRCommandId := udiRCommandId + 1;
                IF udiRCommandId = 0 THEN
                    udiRCommandId := 1;
                END_IF
            END_IF
        END_IF
        IF udiFirstFaultId > 0 THEN
            eExitIntent := CFF_EXIT_FAULT_NO_RETURN;
            eNextState := CFF_EXTSETPOINT_DISABLE;
        ELSIF bStopRequestedLatched OR bAbortEvent OR bResetPendingLatched THEN
            IF fbStepCriterion.stOutput.bEndConfirmed
                AND (fbStepCriterion.stOutput.eEndCause = STEP_END_STOP_REQUEST)
                AND NOT fbForceDecline.stOutput.bFault
                AND NOT fbStepCriterion.stOutput.bFault THEN
                nStepResultIndex := 4;
                bStepResultNok := fbStepCriterion.stOutput.bNok
                    OR (uliQualifiedHold_us < uliQualifiedHoldTarget_us);
                bStepResultPublishRequested := TRUE;
                eEndCause := fbStepCriterion.stOutput.eEndCause;
            END_IF
            eExitIntent := CFF_EXIT_ABORT_NO_RETURN;
            eNextState := CFF_EXTSETPOINT_DISABLE;
        ELSIF NOT bStateEntry
            AND (fbForceDecline.stOutput.bFault OR fbStepCriterion.stOutput.bFault
                OR NOT GVL_Status.stFast.bForceSetpointRampValid
                OR NOT GVL_Status.stFast.bRSpeedRampValid) THEN
            IF udiFirstFaultId = 0 THEN
                udiFirstFaultId := 16#0000A00B;
            END_IF
            eExitIntent := CFF_EXIT_FAULT_NO_RETURN;
            eNextState := CFF_EXTSETPOINT_DISABLE;
        ELSIF NOT bStateEntry AND fbStepCriterion.stOutput.bEndConfirmed THEN
            nStepResultIndex := 4;
            bStepResultNok := fbStepCriterion.stOutput.bNok
                OR (uliQualifiedHold_us < uliQualifiedHoldTarget_us);
            bStepResultPublishRequested := TRUE;
            eEndCause := fbStepCriterion.stOutput.eEndCause;
            IF bStepResultNok OR bCycleNokLatched THEN
                bCycleNokLatched := TRUE;
                eExitIntent := CFF_EXIT_NOK_RETURN;
            ELSE
                eExitIntent := CFF_EXIT_NORMAL_RETURN;
            END_IF
            eNextState := CFF_CONTROLLED_FORCE_UNLOAD;
        ELSIF NOT bStateEntry AND tonStep4RAxisStop.Q THEN
            IF udiFirstFaultId = 0 THEN
                udiFirstFaultId := 16#0000A014;
            END_IF
            eExitIntent := CFF_EXIT_FAULT_NO_RETURN;
            eNextState := CFF_EXTSETPOINT_DISABLE;
        ELSIF NOT bStateEntry
            AND (GVL_Status.stFast.udiAcceptedSequenceRCommandId = udiRCommandId)
            AND GVL_Status.stFast.bRSpeedRampValid
            AND GVL_Status.stFast.bRSpeedRampReached
            AND GVL_Status.stFast.bForceSetpointRampValid
            AND GVL_Status.stFast.bForceSetpointRampReached THEN
            eNextState := CFF_STEP4_VALID_FORCE_HOLD;
        END_IF

    (* Step4 Hold：继续同一Criterion、总时间和暂停式Qualified Hold。 *)
    CFF_STEP4_VALID_FORCE_HOLD:
        stMotionIntent.stZCommand.bEnable := TRUE;
        stMotionIntent.stZCommand.bUseExternalSetpoint := TRUE;
        stMotionIntent.stZCommand.eOwnerRequest := Z_OWNER_FORCE_PROCESS;
        stMotionIntent.bExternalEnableRequest := TRUE;
        stMotionIntent.bRAxisProcessRequested := TRUE;
        stMotionIntent.stRCommand := stLastPublishedRCommand;
        bForceControlEnable := TRUE;
        eStep := CFF_STEP4_COMPRESSION;
        eSubPhase := STEP_SUBPHASE_VALID_FORCE_HOLD;
        IF udiFirstFaultId > 0 THEN
            eExitIntent := CFF_EXIT_FAULT_NO_RETURN;
            eNextState := CFF_EXTSETPOINT_DISABLE;
        ELSIF bStopRequestedLatched OR bAbortEvent OR bResetPendingLatched THEN
            IF fbStepCriterion.stOutput.bEndConfirmed
                AND (fbStepCriterion.stOutput.eEndCause = STEP_END_STOP_REQUEST)
                AND NOT fbForceDecline.stOutput.bFault
                AND NOT fbStepCriterion.stOutput.bFault THEN
                nStepResultIndex := 4;
                bStepResultNok := fbStepCriterion.stOutput.bNok
                    OR (uliQualifiedHold_us < uliQualifiedHoldTarget_us);
                bStepResultPublishRequested := TRUE;
                eEndCause := fbStepCriterion.stOutput.eEndCause;
            END_IF
            eExitIntent := CFF_EXIT_ABORT_NO_RETURN;
            eNextState := CFF_EXTSETPOINT_DISABLE;
        ELSIF fbForceDecline.stOutput.bFault OR fbStepCriterion.stOutput.bFault
            OR NOT GVL_Status.stFast.bForceSetpointRampValid
            OR NOT GVL_Status.stFast.bRSpeedRampValid THEN
            IF udiFirstFaultId = 0 THEN
                udiFirstFaultId := 16#0000A00B;
            END_IF
            eExitIntent := CFF_EXIT_FAULT_NO_RETURN;
            eNextState := CFF_EXTSETPOINT_DISABLE;
        ELSIF fbStepCriterion.stOutput.bEndConfirmed THEN
            nStepResultIndex := 4;
            bStepResultNok := fbStepCriterion.stOutput.bNok
                OR (uliQualifiedHold_us < uliQualifiedHoldTarget_us);
            bStepResultPublishRequested := TRUE;
            eEndCause := fbStepCriterion.stOutput.eEndCause;
            IF bStepResultNok OR bCycleNokLatched THEN
                bCycleNokLatched := TRUE;
                eExitIntent := CFF_EXIT_NOK_RETURN;
            ELSE
                eExitIntent := CFF_EXIT_NORMAL_RETURN;
            END_IF
            eNextState := CFF_CONTROLLED_FORCE_UNLOAD;
        ELSIF tonStep4RAxisStop.Q THEN
            IF udiFirstFaultId = 0 THEN
                udiFirstFaultId := 16#0000A014;
            END_IF
            eExitIntent := CFF_EXIT_FAULT_NO_RETURN;
            eNextState := CFF_EXTSETPOINT_DISABLE;
        END_IF

    CFF_CONTROLLED_FORCE_UNLOAD:
        stMotionIntent.stZCommand.bEnable := TRUE;
        stMotionIntent.stZCommand.bUseExternalSetpoint := TRUE;
        stMotionIntent.stZCommand.eOwnerRequest := Z_OWNER_FORCE_PROCESS;
        stMotionIntent.bExternalEnableRequest := TRUE;
        stMotionIntent.bExternalDisableRequest := FALSE;
        stMotionIntent.rExternalTargetVelocity_mm_s := 0.0;
        stMotionIntent.bForceProcessExitComplete := FALSE;
        stMotionIntent.bRAxisProcessRequested := TRUE;
        rForceSet_kN := 0.0;
        bForceControlEnable := TRUE;
        stMotionIntent.stRCommand.bEnable := TRUE;
        stMotionIntent.stRCommand.bReset := FALSE;
        stMotionIntent.stRCommand.bStop := TRUE;
        stMotionIntent.stRCommand.bMoveVelocity := FALSE;
        stMotionIntent.stRCommand.rVelocity_rpm := 0.0;
        stMotionIntent.stRCommand.rAcceleration_rpm_s := stRAxisProfileSnapshot.fSpeedRampRpmS;
        stMotionIntent.stRCommand.rDeceleration_rpm_s := stRAxisProfileSnapshot.fSpeedRampRpmS;
        IF bStateEntry THEN
            IF NOT bUnloadTransferInitialized AND bUnloadHealthy THEN
                rTargetRelativePosition_mm := GVL_Process.stActual.fSRelSensorMm;
                rForceTransferVelocity_mm_s :=
                    GVL_Status.stFast.stZExtSetpoint.rAcceptedVelocity_mm_s;
                bForceProfileTransferPending := TRUE;
                bUnloadTransferInitialized := TRUE;
            END_IF
            bSafeExitRStopPending := TRUE;
            IF bRCommandPayloadChanged THEN
                stLastPublishedRCommand := stCandidateRCommand;
                stMotionIntent.stRCommand := stCandidateRCommand;
                udiRCommandId := udiRCommandId + 1;
                IF udiRCommandId = 0 THEN
                    udiRCommandId := 1;
                END_IF
            END_IF
        END_IF
        IF bSafeExitRStopPending
            AND (GVL_Status.stFast.udiAcceptedSequenceRCommandId = udiRCommandId)
            AND GVL_Status.stFast.stRAxis.bStandstill THEN
            bSafeExitRStopPending := FALSE;
        END_IF
        (* 卸载条件已成立但连续确认时间未到时，显式保持当前状态。 *)
        IF GVL_Status.stFast.bForceSetpointRampValid
            AND GVL_Status.stFast.bForceSetpointRampReached
            AND ABS(GVL_Process.stActual.fForceControlN)
                <= stCycleSnapshot.stProgram.stHeader.fContactForceOffN
            AND ABS(GVL_Status.stFast.stZExtSetpoint.rAcceptedVelocity_mm_s)
                <= stZExtConfigSnapshot.rStandstillVelocity_mm_s
            AND bUnloadHealthy
            AND (tonUnloadStandstillConfirm.ET
                < stSequenceConfigSnapshot.tUnloadStandstillConfirm) THEN
            eNextState := eState;
        END_IF
        IF tonControlledUnload.ET
            < stSequenceConfigSnapshot.tControlledUnloadTimeout THEN
            eNextState := eState;
        END_IF
        IF udiFirstFaultId > 0 THEN
            eExitIntent := CFF_EXIT_FAULT_NO_RETURN;
            eNextState := CFF_EXTSETPOINT_DISABLE;
        ELSIF tonControlledUnload.Q THEN
            IF udiFirstFaultId = 0 THEN
                udiFirstFaultId := 16#0000A013;
            END_IF
            eExitIntent := CFF_EXIT_FAULT_NO_RETURN;
            eNextState := CFF_EXTSETPOINT_DISABLE;
        ELSIF tonUnloadStandstillConfirm.Q THEN
            eNextState := CFF_EXTSETPOINT_DISABLE;
        END_IF

    CFF_EXTSETPOINT_DISABLE:
        stMotionIntent.stZCommand.bEnable := TRUE;
        stMotionIntent.stZCommand.bUseExternalSetpoint := TRUE;
        stMotionIntent.stZCommand.eOwnerRequest := Z_OWNER_FORCE_PROCESS;
        stMotionIntent.stZCommand.rDeceleration_mm_s2 :=
            stSequenceConfigSnapshot.fStandardMoveDecelerationMmS2;
        stMotionIntent.bExternalEnableRequest := FALSE;
        stMotionIntent.bExternalDisableRequest := TRUE;
        stMotionIntent.rExternalTargetVelocity_mm_s := 0.0;
        stMotionIntent.bForceProcessExitComplete := FALSE;
        stMotionIntent.bRAxisProcessRequested := TRUE;
        stMotionIntent.stRCommand.bEnable := TRUE;
        stMotionIntent.stRCommand.bReset := FALSE;
        stMotionIntent.stRCommand.bStop := TRUE;
        stMotionIntent.stRCommand.bMoveVelocity := FALSE;
        stMotionIntent.stRCommand.rVelocity_rpm := 0.0;
        stMotionIntent.stRCommand.rAcceleration_rpm_s := stRAxisProfileSnapshot.fSpeedRampRpmS;
        stMotionIntent.stRCommand.rDeceleration_rpm_s := stRAxisProfileSnapshot.fSpeedRampRpmS;
        bForceControlEnable := FALSE;
        IF bUnknownExternalRStopPending
            AND (GVL_Status.stFast.udiAcceptedSequenceRCommandId = udiRCommandId)
            AND GVL_Status.stFast.stRAxis.bStandstill THEN
            bUnknownExternalRStopPending := FALSE;
        END_IF
        IF bSafeExitRStopPending
            AND (GVL_Status.stFast.udiAcceptedSequenceRCommandId = udiRCommandId)
            AND GVL_Status.stFast.stRAxis.bStandstill THEN
            bSafeExitRStopPending := FALSE;
        END_IF
        IF GVL_Status.stFast.stZExtSetpoint.bReleaseOwner
            AND NOT bUnknownExternalRStopPending
            AND NOT bSafeExitRStopPending
            AND (GVL_Status.stFast.udiAcceptedSequenceRCommandId = udiRCommandId)
            AND GVL_Status.stFast.stRAxis.bStandstill THEN
            stMotionIntent.bForceProcessExitComplete := TRUE;
            IF udiFirstFaultId > 0 THEN
                eExitIntent := CFF_EXIT_FAULT_NO_RETURN;
                eNextState := CFF_FAULT;
            ELSIF bStopRequestedLatched OR bAbortEvent OR bResetPendingLatched THEN
                eExitIntent := CFF_EXIT_ABORT_NO_RETURN;
                eNextState := CFF_ABORT;
            ELSE
                CASE eExitIntent OF
                    CFF_EXIT_NORMAL_RETURN:
                        IF GVL_Status.stFast.stZAxis.bReady
                            AND GVL_Status.stFast.stRAxis.bReady
                            AND NOT GVL_Status.stFast.stZAxis.bError
                            AND NOT GVL_Status.stFast.stRAxis.bError THEN
                            IF stCycleSnapshot.stProgram.stHeader.eReturnMode = RETURN_MODE_LOCAL THEN
                                eNextState := CFF_RETURN_LOCAL;
                            ELSIF stCycleSnapshot.stProgram.stHeader.eReturnMode = RETURN_MODE_REFERENCE THEN
                                eNextState := CFF_RETURN_REFERENCE;
                            ELSE
                                IF udiFirstFaultId = 0 THEN
                                    udiFirstFaultId := 16#0000A016;
                                END_IF
                                eExitIntent := CFF_EXIT_FAULT_NO_RETURN;
                                eNextState := CFF_FAULT;
                            END_IF
                        ELSE
                            IF udiFirstFaultId = 0 THEN
                                udiFirstFaultId := 16#0000A016;
                            END_IF
                            eExitIntent := CFF_EXIT_FAULT_NO_RETURN;
                            eNextState := CFF_FAULT;
                        END_IF
                    CFF_EXIT_NOK_RETURN:
                        IF GVL_Status.stFast.stZAxis.bReady
                            AND GVL_Status.stFast.stRAxis.bReady
                            AND NOT GVL_Status.stFast.stZAxis.bError
                            AND NOT GVL_Status.stFast.stRAxis.bError THEN
                            IF stCycleSnapshot.stProgram.stHeader.eReturnMode = RETURN_MODE_LOCAL THEN
                                eNextState := CFF_RETURN_LOCAL;
                            ELSIF stCycleSnapshot.stProgram.stHeader.eReturnMode = RETURN_MODE_REFERENCE THEN
                                eNextState := CFF_RETURN_REFERENCE;
                            ELSE
                                IF udiFirstFaultId = 0 THEN
                                    udiFirstFaultId := 16#0000A016;
                                END_IF
                                eExitIntent := CFF_EXIT_FAULT_NO_RETURN;
                                eNextState := CFF_FAULT;
                            END_IF
                        ELSE
                            IF udiFirstFaultId = 0 THEN
                                udiFirstFaultId := 16#0000A016;
                            END_IF
                            eExitIntent := CFF_EXIT_FAULT_NO_RETURN;
                            eNextState := CFF_FAULT;
                        END_IF
                    CFF_EXIT_ABORT_NO_RETURN:
                        eNextState := CFF_ABORT;
                    CFF_EXIT_FAULT_NO_RETURN:
                        eNextState := CFF_FAULT;
                ELSE
                    IF udiFirstFaultId = 0 THEN
                        udiFirstFaultId := 16#0000A016;
                    END_IF
                    eExitIntent := CFF_EXIT_FAULT_NO_RETURN;
                    eNextState := CFF_FAULT;
                END_CASE
            END_IF
            IF (eNextState = CFF_ABORT) OR (eNextState = CFF_FAULT) THEN
                bTerminalFaultStopRequired := TRUE;
            END_IF
        END_IF

    CFF_RETURN_LOCAL:
        IF NOT bReturnEntryBlocked THEN
            IF bReturnPublicationAllowed THEN
                IF bStateEntry THEN
                    udiZCommandId := udiZCommandId + 1;
                    IF udiZCommandId = 0 THEN
                        udiZCommandId := 1;
                    END_IF
                END_IF
                stMotionIntent.stZCommand.bEnable := TRUE;
                stMotionIntent.stZCommand.bReset := FALSE;
                stMotionIntent.stZCommand.bStop := FALSE;
                stMotionIntent.stZCommand.bHome := FALSE;
                stMotionIntent.stZCommand.bMoveAbsolute := TRUE;
                stMotionIntent.stZCommand.bMoveVelocity := FALSE;
                stMotionIntent.stZCommand.bUseExternalSetpoint := FALSE;
                stMotionIntent.stZCommand.rHomePosition_mm := 0.0;
                stMotionIntent.stZCommand.rPosition_mm := rCycleStartZPosition_mm;
                stMotionIntent.stZCommand.rVelocity_mm_s :=
                    stCycleSnapshot.stProgram.stHeader.fReturnVelocityMmS;
                stMotionIntent.stZCommand.rAcceleration_mm_s2 :=
                    stSequenceConfigSnapshot.fStandardMoveAccelerationMmS2;
                stMotionIntent.stZCommand.rDeceleration_mm_s2 :=
                    stSequenceConfigSnapshot.fStandardMoveDecelerationMmS2;
                stMotionIntent.stZCommand.eOwnerRequest := Z_OWNER_RETRACT;
                stMotionIntent.bExternalEnableRequest := FALSE;
                stMotionIntent.bExternalDisableRequest := FALSE;
                stMotionIntent.rExternalTargetVelocity_mm_s := 0.0;
                stMotionIntent.bForceProcessExitComplete := TRUE;
                stMotionIntent.bRAxisProcessRequested := TRUE;
                stMotionIntent.stRCommand.bEnable := TRUE;
                stMotionIntent.stRCommand.bReset := FALSE;
                stMotionIntent.stRCommand.bStop := TRUE;
                stMotionIntent.stRCommand.bMoveVelocity := FALSE;
                stMotionIntent.stRCommand.rVelocity_rpm := 0.0;
                stMotionIntent.stRCommand.rAcceleration_rpm_s :=
                    stRAxisProfileSnapshot.fSpeedRampRpmS;
                stMotionIntent.stRCommand.rDeceleration_rpm_s :=
                    stRAxisProfileSnapshot.fSpeedRampRpmS;
                bForceControlEnable := FALSE;
                IF tonReturn.Q THEN
                    IF udiFirstFaultId = 0 THEN
                        udiFirstFaultId := 16#0000A015;
                    END_IF
                    eExitIntent := CFF_EXIT_FAULT_NO_RETURN;
                    eNextState := CFF_FAULT;
                END_IF
                IF (GVL_Status.stFast.udiAcceptedSequenceZCommandId = udiZCommandId)
                    AND GVL_Status.stFast.stZAxis.bDone
                    AND GVL_Status.stFast.stZAxis.bStandstill
                    AND NOT tonReturn.Q THEN
                    eNextState := CFF_EVALUATE;
                END_IF
            ELSE
                IF udiFirstFaultId = 0 THEN
                    udiFirstFaultId := 16#0000A016;
                END_IF
                eExitIntent := CFF_EXIT_FAULT_NO_RETURN;
                eNextState := CFF_FAULT;
            END_IF
        END_IF
    CFF_RETURN_REFERENCE:
        IF NOT bReturnEntryBlocked THEN
            IF bReturnPublicationAllowed THEN
                IF bStateEntry THEN
                    udiZCommandId := udiZCommandId + 1;
                    IF udiZCommandId = 0 THEN
                        udiZCommandId := 1;
                    END_IF
                END_IF
                stMotionIntent.stZCommand.bEnable := TRUE;
                stMotionIntent.stZCommand.bReset := FALSE;
                stMotionIntent.stZCommand.bStop := FALSE;
                stMotionIntent.stZCommand.bHome := FALSE;
                stMotionIntent.stZCommand.bMoveAbsolute := TRUE;
                stMotionIntent.stZCommand.bMoveVelocity := FALSE;
                stMotionIntent.stZCommand.bUseExternalSetpoint := FALSE;
                stMotionIntent.stZCommand.rHomePosition_mm := 0.0;
                stMotionIntent.stZCommand.rPosition_mm :=
                    stCycleSnapshot.stProgram.stHeader.fReturnOpeningMm;
                stMotionIntent.stZCommand.rVelocity_mm_s :=
                    stCycleSnapshot.stProgram.stHeader.fReturnVelocityMmS;
                stMotionIntent.stZCommand.rAcceleration_mm_s2 :=
                    stSequenceConfigSnapshot.fStandardMoveAccelerationMmS2;
                stMotionIntent.stZCommand.rDeceleration_mm_s2 :=
                    stSequenceConfigSnapshot.fStandardMoveDecelerationMmS2;
                stMotionIntent.stZCommand.eOwnerRequest := Z_OWNER_RETRACT;
                stMotionIntent.bExternalEnableRequest := FALSE;
                stMotionIntent.bExternalDisableRequest := FALSE;
                stMotionIntent.rExternalTargetVelocity_mm_s := 0.0;
                stMotionIntent.bForceProcessExitComplete := TRUE;
                stMotionIntent.bRAxisProcessRequested := TRUE;
                stMotionIntent.stRCommand.bEnable := TRUE;
                stMotionIntent.stRCommand.bReset := FALSE;
                stMotionIntent.stRCommand.bStop := TRUE;
                stMotionIntent.stRCommand.bMoveVelocity := FALSE;
                stMotionIntent.stRCommand.rVelocity_rpm := 0.0;
                stMotionIntent.stRCommand.rAcceleration_rpm_s :=
                    stRAxisProfileSnapshot.fSpeedRampRpmS;
                stMotionIntent.stRCommand.rDeceleration_rpm_s :=
                    stRAxisProfileSnapshot.fSpeedRampRpmS;
                bForceControlEnable := FALSE;
                IF tonReturn.Q THEN
                    IF udiFirstFaultId = 0 THEN
                        udiFirstFaultId := 16#0000A015;
                    END_IF
                    eExitIntent := CFF_EXIT_FAULT_NO_RETURN;
                    eNextState := CFF_FAULT;
                END_IF
                IF (GVL_Status.stFast.udiAcceptedSequenceZCommandId = udiZCommandId)
                    AND GVL_Status.stFast.stZAxis.bDone
                    AND GVL_Status.stFast.stZAxis.bStandstill
                    AND NOT tonReturn.Q THEN
                    eNextState := CFF_EVALUATE;
                END_IF
            ELSE
                IF udiFirstFaultId = 0 THEN
                    udiFirstFaultId := 16#0000A016;
                END_IF
                eExitIntent := CFF_EXIT_FAULT_NO_RETURN;
                eNextState := CFF_FAULT;
            END_IF
        END_IF
    CFF_EVALUATE:
        stMotionIntent.stZCommand.bEnable := TRUE;
        stMotionIntent.stZCommand.bReset := FALSE;
        stMotionIntent.stZCommand.bStop := FALSE;
        stMotionIntent.stZCommand.bHome := FALSE;
        stMotionIntent.stZCommand.bMoveAbsolute := TRUE;
        stMotionIntent.stZCommand.bMoveVelocity := FALSE;
        stMotionIntent.stZCommand.bUseExternalSetpoint := FALSE;
        stMotionIntent.stZCommand.rHomePosition_mm := 0.0;
        stMotionIntent.stZCommand.rPosition_mm := SEL(
            stCycleSnapshot.stProgram.stHeader.eReturnMode = RETURN_MODE_REFERENCE,
            rCycleStartZPosition_mm,
            stCycleSnapshot.stProgram.stHeader.fReturnOpeningMm);
        stMotionIntent.stZCommand.rVelocity_mm_s :=
            stCycleSnapshot.stProgram.stHeader.fReturnVelocityMmS;
        stMotionIntent.stZCommand.rAcceleration_mm_s2 :=
            stSequenceConfigSnapshot.fStandardMoveAccelerationMmS2;
        stMotionIntent.stZCommand.rDeceleration_mm_s2 :=
            stSequenceConfigSnapshot.fStandardMoveDecelerationMmS2;
        stMotionIntent.stZCommand.eOwnerRequest := Z_OWNER_RETRACT;
        stMotionIntent.bExternalEnableRequest := FALSE;
        stMotionIntent.bExternalDisableRequest := FALSE;
        stMotionIntent.rExternalTargetVelocity_mm_s := 0.0;
        stMotionIntent.bForceProcessExitComplete := TRUE;
        stMotionIntent.bRAxisProcessRequested := TRUE;
        stMotionIntent.stRCommand.bEnable := TRUE;
        stMotionIntent.stRCommand.bReset := FALSE;
        stMotionIntent.stRCommand.bStop := TRUE;
        stMotionIntent.stRCommand.bMoveVelocity := FALSE;
        stMotionIntent.stRCommand.rVelocity_rpm := 0.0;
        stMotionIntent.stRCommand.rAcceleration_rpm_s := stRAxisProfileSnapshot.fSpeedRampRpmS;
        stMotionIntent.stRCommand.rDeceleration_rpm_s := stRAxisProfileSnapshot.fSpeedRampRpmS;
        bForceControlEnable := FALSE;
        nWrittenStepPrefix := 0;
        bStepResultHole := FALSE;
        bMissingStepResult := FALSE;
        bEvaluateNok := FALSE;
        bEvaluateFault := FALSE;
        FOR nStepIndex := 1 TO 4 DO
            IF abStepResultWritten[nStepIndex] THEN
                IF NOT bMissingStepResult THEN
                    nWrittenStepPrefix := nStepIndex;
                END_IF
                IF bMissingStepResult THEN
                    bStepResultHole := TRUE;
                END_IF
                bEvaluateNok := bEvaluateNok
                    OR GVL_Process.astStepCriterion[nStepIndex].bNok
                    OR GVL_Process.astStepCriterion[nStepIndex].bTooShort
                    OR GVL_Process.astStepCriterion[nStepIndex].bSecondaryLatched
                    OR (GVL_Process.astStepCriterion[nStepIndex].eEndCause
                        = STEP_END_MAX_TIME);
            ELSE
                bMissingStepResult := TRUE;
            END_IF
        END_FOR
        IF abStepResultWritten[4] THEN
            bEvaluateNok := bEvaluateNok
                OR NOT GVL_Process.astStepCriterion[4].bQualifiedForceHoldMet;
        END_IF
        bEvaluateFault := bStepResultHole;
        IF eExitIntent = CFF_EXIT_NORMAL_RETURN THEN
            IF (nWrittenStepPrefix <> 4) OR bEvaluateNok THEN
                bEvaluateFault := TRUE;
            END_IF
        ELSIF eExitIntent = CFF_EXIT_NOK_RETURN THEN
            IF NOT ((nWrittenStepPrefix >= 1) AND bEvaluateNok) THEN
                bEvaluateFault := TRUE;
            END_IF
        ELSIF eExitIntent = CFF_EXIT_ABORT_NO_RETURN THEN
            bEvaluateFault := FALSE;
        ELSE
            bEvaluateFault := TRUE;
        END_IF
        IF bEvaluateFault THEN
            IF udiFirstFaultId = 0 THEN
                udiFirstFaultId := 16#0000A016;
            END_IF
            eExitIntent := CFF_EXIT_FAULT_NO_RETURN;
        END_IF
        IF (eExitIntent = CFF_EXIT_NORMAL_RETURN) AND NOT bEvaluateFault THEN
            eNextState := CFF_COMPLETE_OK;
        ELSIF (eExitIntent = CFF_EXIT_NOK_RETURN) AND NOT bEvaluateFault THEN
            eNextState := CFF_COMPLETE_NOK;
        ELSIF (eExitIntent = CFF_EXIT_ABORT_NO_RETURN) AND NOT bEvaluateFault THEN
            eNextState := CFF_ABORT;
        ELSE
            eNextState := CFF_FAULT;
        END_IF
    CFF_COMPLETE_OK:
        stMotionIntent.stZCommand.bEnable := TRUE;
        stMotionIntent.stZCommand.bReset := FALSE;
        stMotionIntent.stZCommand.bStop := FALSE;
        stMotionIntent.stZCommand.bHome := FALSE;
        stMotionIntent.stZCommand.bMoveAbsolute := TRUE;
        stMotionIntent.stZCommand.bMoveVelocity := FALSE;
        stMotionIntent.stZCommand.bUseExternalSetpoint := FALSE;
        stMotionIntent.stZCommand.rHomePosition_mm := 0.0;
        stMotionIntent.stZCommand.rPosition_mm := SEL(
            stCycleSnapshot.stProgram.stHeader.eReturnMode = RETURN_MODE_REFERENCE,
            rCycleStartZPosition_mm,
            stCycleSnapshot.stProgram.stHeader.fReturnOpeningMm);
        stMotionIntent.stZCommand.rVelocity_mm_s :=
            stCycleSnapshot.stProgram.stHeader.fReturnVelocityMmS;
        stMotionIntent.stZCommand.rAcceleration_mm_s2 :=
            stSequenceConfigSnapshot.fStandardMoveAccelerationMmS2;
        stMotionIntent.stZCommand.rDeceleration_mm_s2 :=
            stSequenceConfigSnapshot.fStandardMoveDecelerationMmS2;
        stMotionIntent.stZCommand.eOwnerRequest := Z_OWNER_RETRACT;
        stMotionIntent.bExternalEnableRequest := FALSE;
        stMotionIntent.bExternalDisableRequest := FALSE;
        stMotionIntent.rExternalTargetVelocity_mm_s := 0.0;
        stMotionIntent.bForceProcessExitComplete := TRUE;
        stMotionIntent.bRAxisProcessRequested := TRUE;
        stMotionIntent.stRCommand.bEnable := TRUE;
        stMotionIntent.stRCommand.bReset := FALSE;
        stMotionIntent.stRCommand.bStop := TRUE;
        stMotionIntent.stRCommand.bMoveVelocity := FALSE;
        stMotionIntent.stRCommand.rVelocity_rpm := 0.0;
        stMotionIntent.stRCommand.rAcceleration_rpm_s := stRAxisProfileSnapshot.fSpeedRampRpmS;
        stMotionIntent.stRCommand.rDeceleration_rpm_s := stRAxisProfileSnapshot.fSpeedRampRpmS;
        bForceControlEnable := FALSE;
        IF GVL_Status.stFast.stZAxis.bStandstill
            AND GVL_Status.stFast.stRAxis.bStandstill
            AND bExternalReady THEN
            bBusy := FALSE;
            bDone := TRUE;
            bError := FALSE;
            bAborted := FALSE;
        END_IF
    CFF_COMPLETE_NOK:
        stMotionIntent.stZCommand.bEnable := TRUE;
        stMotionIntent.stZCommand.bReset := FALSE;
        stMotionIntent.stZCommand.bStop := FALSE;
        stMotionIntent.stZCommand.bHome := FALSE;
        stMotionIntent.stZCommand.bMoveAbsolute := TRUE;
        stMotionIntent.stZCommand.bMoveVelocity := FALSE;
        stMotionIntent.stZCommand.bUseExternalSetpoint := FALSE;
        stMotionIntent.stZCommand.rHomePosition_mm := 0.0;
        stMotionIntent.stZCommand.rPosition_mm := SEL(
            stCycleSnapshot.stProgram.stHeader.eReturnMode = RETURN_MODE_REFERENCE,
            rCycleStartZPosition_mm,
            stCycleSnapshot.stProgram.stHeader.fReturnOpeningMm);
        stMotionIntent.stZCommand.rVelocity_mm_s :=
            stCycleSnapshot.stProgram.stHeader.fReturnVelocityMmS;
        stMotionIntent.stZCommand.rAcceleration_mm_s2 :=
            stSequenceConfigSnapshot.fStandardMoveAccelerationMmS2;
        stMotionIntent.stZCommand.rDeceleration_mm_s2 :=
            stSequenceConfigSnapshot.fStandardMoveDecelerationMmS2;
        stMotionIntent.stZCommand.eOwnerRequest := Z_OWNER_RETRACT;
        stMotionIntent.bExternalEnableRequest := FALSE;
        stMotionIntent.bExternalDisableRequest := FALSE;
        stMotionIntent.rExternalTargetVelocity_mm_s := 0.0;
        stMotionIntent.bForceProcessExitComplete := TRUE;
        stMotionIntent.bRAxisProcessRequested := TRUE;
        stMotionIntent.stRCommand.bEnable := TRUE;
        stMotionIntent.stRCommand.bReset := FALSE;
        stMotionIntent.stRCommand.bStop := TRUE;
        stMotionIntent.stRCommand.bMoveVelocity := FALSE;
        stMotionIntent.stRCommand.rVelocity_rpm := 0.0;
        stMotionIntent.stRCommand.rAcceleration_rpm_s := stRAxisProfileSnapshot.fSpeedRampRpmS;
        stMotionIntent.stRCommand.rDeceleration_rpm_s := stRAxisProfileSnapshot.fSpeedRampRpmS;
        bForceControlEnable := FALSE;
        IF GVL_Status.stFast.stZAxis.bStandstill
            AND GVL_Status.stFast.stRAxis.bStandstill
            AND bExternalReady THEN
            bBusy := FALSE;
            bDone := TRUE;
            bError := TRUE;
            bAborted := FALSE;
        END_IF
    CFF_ABORT:
        IF bStateEntry AND bTerminalFaultStopRequired
            AND NOT bApproachFaultStopPending THEN
            udiZCommandId := udiZCommandId + 1;
            IF udiZCommandId = 0 THEN
                udiZCommandId := 1;
            END_IF
            bApproachFaultStopPending := TRUE;
            bTerminalFaultStopRequired := FALSE;
        END_IF
        stMotionIntent.stZCommand.bEnable := TRUE;
        stMotionIntent.stZCommand.bReset := FALSE;
        stMotionIntent.stZCommand.bStop := TRUE;
        stMotionIntent.stZCommand.bHome := FALSE;
        stMotionIntent.stZCommand.bMoveAbsolute := FALSE;
        stMotionIntent.stZCommand.bMoveVelocity := FALSE;
        stMotionIntent.stZCommand.bUseExternalSetpoint := FALSE;
        stMotionIntent.stZCommand.rHomePosition_mm := 0.0;
        stMotionIntent.stZCommand.rPosition_mm := 0.0;
        stMotionIntent.stZCommand.rVelocity_mm_s := 0.0;
        stMotionIntent.stZCommand.rAcceleration_mm_s2 := stSequenceConfigSnapshot.fStandardMoveAccelerationMmS2;
        stMotionIntent.stZCommand.rDeceleration_mm_s2 := stSequenceConfigSnapshot.fStandardMoveDecelerationMmS2;
        stMotionIntent.stZCommand.eOwnerRequest := Z_OWNER_FAULT_STOP;
        stMotionIntent.bExternalEnableRequest := FALSE;
        stMotionIntent.bExternalDisableRequest := FALSE;
        stMotionIntent.rExternalTargetVelocity_mm_s := 0.0;
        stMotionIntent.bForceProcessExitComplete := TRUE;
        stMotionIntent.bRAxisProcessRequested := TRUE;
        stMotionIntent.stRCommand.bEnable := TRUE;
        stMotionIntent.stRCommand.bReset := FALSE;
        stMotionIntent.stRCommand.bStop := TRUE;
        stMotionIntent.stRCommand.bMoveVelocity := FALSE;
        stMotionIntent.stRCommand.rVelocity_rpm := 0.0;
        stMotionIntent.stRCommand.rAcceleration_rpm_s := stRAxisProfileSnapshot.fSpeedRampRpmS;
        stMotionIntent.stRCommand.rDeceleration_rpm_s := stRAxisProfileSnapshot.fSpeedRampRpmS;
        bForceControlEnable := FALSE;
        IF bApproachFaultStopPending
            AND (GVL_Status.stFast.udiAcceptedSequenceZCommandId = udiZCommandId)
            AND GVL_Status.stFast.stZAxis.bStandstill
            AND (GVL_Status.stFast.udiAcceptedSequenceRCommandId = udiRCommandId)
            AND GVL_Status.stFast.stRAxis.bStandstill THEN
            bApproachFaultStopPending := FALSE;
        END_IF
        IF NOT bApproachFaultStopPending
            AND GVL_Status.stFast.stZAxis.bStandstill
            AND GVL_Status.stFast.stRAxis.bStandstill
            AND bExternalReady THEN
            bBusy := FALSE;
            bDone := FALSE;
            bError := FALSE;
            bAborted := TRUE;
        END_IF
    CFF_FAULT:
        IF udiFirstFaultId = 0 THEN
            udiFirstFaultId := 16#0000A016;
        END_IF
        IF bStateEntry AND bTerminalFaultStopRequired
            AND NOT bApproachFaultStopPending THEN
            udiZCommandId := udiZCommandId + 1;
            IF udiZCommandId = 0 THEN
                udiZCommandId := 1;
            END_IF
            bApproachFaultStopPending := TRUE;
            bTerminalFaultStopRequired := FALSE;
        END_IF
        stMotionIntent.stZCommand.bEnable := TRUE;
        stMotionIntent.stZCommand.bReset := FALSE;
        stMotionIntent.stZCommand.bStop := TRUE;
        stMotionIntent.stZCommand.bHome := FALSE;
        stMotionIntent.stZCommand.bMoveAbsolute := FALSE;
        stMotionIntent.stZCommand.bMoveVelocity := FALSE;
        stMotionIntent.stZCommand.bUseExternalSetpoint := FALSE;
        stMotionIntent.stZCommand.rHomePosition_mm := 0.0;
        stMotionIntent.stZCommand.rPosition_mm := 0.0;
        stMotionIntent.stZCommand.rVelocity_mm_s := 0.0;
        stMotionIntent.stZCommand.rAcceleration_mm_s2 := stSequenceConfigSnapshot.fStandardMoveAccelerationMmS2;
        stMotionIntent.stZCommand.rDeceleration_mm_s2 := stSequenceConfigSnapshot.fStandardMoveDecelerationMmS2;
        stMotionIntent.stZCommand.eOwnerRequest := Z_OWNER_FAULT_STOP;
        stMotionIntent.bExternalEnableRequest := FALSE;
        stMotionIntent.bExternalDisableRequest := FALSE;
        stMotionIntent.rExternalTargetVelocity_mm_s := 0.0;
        stMotionIntent.bForceProcessExitComplete := TRUE;
        stMotionIntent.bRAxisProcessRequested := TRUE;
        stMotionIntent.stRCommand.bEnable := TRUE;
        stMotionIntent.stRCommand.bReset := FALSE;
        stMotionIntent.stRCommand.bStop := TRUE;
        stMotionIntent.stRCommand.bMoveVelocity := FALSE;
        stMotionIntent.stRCommand.rVelocity_rpm := 0.0;
        stMotionIntent.stRCommand.rAcceleration_rpm_s := stRAxisProfileSnapshot.fSpeedRampRpmS;
        stMotionIntent.stRCommand.rDeceleration_rpm_s := stRAxisProfileSnapshot.fSpeedRampRpmS;
        bForceControlEnable := FALSE;
        IF bApproachFaultStopPending
            AND (GVL_Status.stFast.udiAcceptedSequenceZCommandId = udiZCommandId)
            AND GVL_Status.stFast.stZAxis.bStandstill
            AND (GVL_Status.stFast.udiAcceptedSequenceRCommandId = udiRCommandId)
            AND GVL_Status.stFast.stRAxis.bStandstill THEN
            bApproachFaultStopPending := FALSE;
        END_IF
        IF NOT bApproachFaultStopPending
            AND GVL_Status.stFast.stZAxis.bStandstill
            AND GVL_Status.stFast.stRAxis.bStandstill
            AND bExternalReady THEN
            bBusy := FALSE;
            bDone := FALSE;
            bError := TRUE;
            bAborted := FALSE;
        END_IF
ELSE
    IF udiFirstFaultId = 0 THEN
        udiFirstFaultId := 16#0000A016;
    END_IF
    eExitIntent := CFF_EXIT_FAULT_NO_RETURN;
    IF NOT bExternalReady THEN
        (* Unknown state while External still owns the axis: preserve the
           active Z identity/owner contract and create a fresh R stop. *)
        IF udiZCommandId = 0 THEN
            udiZCommandId := 1;
        END_IF
        udiRCommandId := udiRCommandId + 1;
        IF udiRCommandId = 0 THEN
            udiRCommandId := 1;
        END_IF
        bUnknownExternalRStopPending := TRUE;
        stMotionIntent.stZCommand.bEnable := TRUE;
        stMotionIntent.stZCommand.bReset := FALSE;
        stMotionIntent.stZCommand.bStop := FALSE;
        stMotionIntent.stZCommand.bHome := FALSE;
        stMotionIntent.stZCommand.bMoveAbsolute := FALSE;
        stMotionIntent.stZCommand.bMoveVelocity := FALSE;
        stMotionIntent.stZCommand.eOwnerRequest := Z_OWNER_FORCE_PROCESS;
        stMotionIntent.stZCommand.bUseExternalSetpoint := TRUE;
        stMotionIntent.stZCommand.rHomePosition_mm := 0.0;
        stMotionIntent.stZCommand.rPosition_mm := 0.0;
        stMotionIntent.stZCommand.rVelocity_mm_s := 0.0;
        stMotionIntent.stZCommand.rAcceleration_mm_s2 := 0.0;
        stMotionIntent.stZCommand.rDeceleration_mm_s2 :=
            stSequenceConfigSnapshot.fStandardMoveDecelerationMmS2;
        stMotionIntent.bExternalEnableRequest := FALSE;
        stMotionIntent.bExternalDisableRequest := TRUE;
        stMotionIntent.rExternalTargetVelocity_mm_s := 0.0;
        stMotionIntent.bForceProcessExitComplete := FALSE;
        stMotionIntent.bRAxisProcessRequested := TRUE;
        stMotionIntent.stRCommand.bEnable := TRUE;
        stMotionIntent.stRCommand.bReset := FALSE;
        stMotionIntent.stRCommand.bStop := TRUE;
        stMotionIntent.stRCommand.bMoveVelocity := FALSE;
        stMotionIntent.stRCommand.rVelocity_rpm := 0.0;
        stMotionIntent.stRCommand.rAcceleration_rpm_s := stRAxisProfileSnapshot.fSpeedRampRpmS;
        stMotionIntent.stRCommand.rDeceleration_rpm_s := stRAxisProfileSnapshot.fSpeedRampRpmS;
        bForceControlEnable := FALSE;
        eNextState := CFF_EXTSETPOINT_DISABLE;
    ELSE
        (* External is released, so terminate any possible standard NC motion
           with one fresh FaultStop transaction and retain the R zero-stop. *)
        udiZCommandId := udiZCommandId + 1;
        IF udiZCommandId = 0 THEN
            udiZCommandId := 1;
        END_IF
        udiRCommandId := udiRCommandId + 1;
        IF udiRCommandId = 0 THEN
            udiRCommandId := 1;
        END_IF
        bApproachFaultStopPending := TRUE;
        stMotionIntent.stZCommand.bEnable := TRUE;
        stMotionIntent.stZCommand.bReset := FALSE;
        stMotionIntent.stZCommand.bStop := TRUE;
        stMotionIntent.stZCommand.bHome := FALSE;
        stMotionIntent.stZCommand.bMoveAbsolute := FALSE;
        stMotionIntent.stZCommand.bMoveVelocity := FALSE;
        stMotionIntent.stZCommand.eOwnerRequest := Z_OWNER_FAULT_STOP;
        stMotionIntent.stZCommand.bUseExternalSetpoint := FALSE;
        stMotionIntent.stZCommand.rHomePosition_mm := 0.0;
        stMotionIntent.stZCommand.rPosition_mm := 0.0;
        stMotionIntent.stZCommand.rVelocity_mm_s := 0.0;
        stMotionIntent.stZCommand.rAcceleration_mm_s2 := stSequenceConfigSnapshot.fStandardMoveAccelerationMmS2;
        stMotionIntent.stZCommand.rDeceleration_mm_s2 := stSequenceConfigSnapshot.fStandardMoveDecelerationMmS2;
        stMotionIntent.bExternalEnableRequest := FALSE;
        stMotionIntent.bExternalDisableRequest := FALSE;
        stMotionIntent.rExternalTargetVelocity_mm_s := 0.0;
        stMotionIntent.bRAxisProcessRequested := TRUE;
        stMotionIntent.stRCommand.bEnable := TRUE;
        stMotionIntent.stRCommand.bReset := FALSE;
        stMotionIntent.stRCommand.bStop := TRUE;
        stMotionIntent.stRCommand.bMoveVelocity := FALSE;
        stMotionIntent.stRCommand.rVelocity_rpm := 0.0;
        stMotionIntent.stRCommand.rAcceleration_rpm_s := stRAxisProfileSnapshot.fSpeedRampRpmS;
        stMotionIntent.stRCommand.rDeceleration_rpm_s := stRAxisProfileSnapshot.fSpeedRampRpmS;
        bForceControlEnable := FALSE;
        eNextState := CFF_FAULT;
    END_IF
END_CASE

(* 唯一结果发布点：先构造完整payload，再写公开槽位，最后锁存guard。 *)
IF bStepResultPublishRequested AND NOT abStepResultWritten[nStepResultIndex] THEN
    stStepResultCandidate := stClearedStepCriterionResult;
    stStepResultCandidate.eStep := eStep;
    stStepResultCandidate.eEndCause := fbStepCriterion.stOutput.eEndCause;
    stStepResultCandidate.bPrimaryLatched := fbStepCriterion.stOutput.bPrimaryMet;
    stStepResultCandidate.bSecondaryLatched :=
        fbStepCriterion.stOutput.bSecondaryLimitReached;
    stStepResultCandidate.bNok := bStepResultNok;
    stStepResultCandidate.nTriggerCycle := GVL_Status.stFast.nCycleCounter;
    stStepResultCandidate.bTooShort := fbStepCriterion.stOutput.bTooShort;
    stStepResultCandidate.bQualifiedForceHoldMet := (nStepResultIndex = 4)
        AND (uliQualifiedHold_us >= uliQualifiedHoldTarget_us);
    stStepResultCandidate.rQualifiedForceHoldTime_s := rQualifiedForceHoldTime_s;
    stStepResultCandidate.rLatchedForce_kN :=
        fbStepCriterion.stOutput.rLatchedForce_kN;
    stStepResultCandidate.rLatchedRelativePosition_mm :=
        fbStepCriterion.stOutput.rLatchedRelativePosition_mm;
    stStepResultCandidate.rLatchedStepTime_s :=
        fbStepCriterion.stOutput.rLatchedStepTime_s;
    GVL_Process.astStepCriterion[nStepResultIndex] := stStepResultCandidate;
    abStepResultWritten[nStepResultIndex] := TRUE;
END_IF

(* This classifier is evaluated after the state branch so a newly latched
   timeout/algorithm fault is routed to safety in the same Fast scan. *)
bSafeExitRequested := bStopRequestedLatched OR bAbortEvent OR bResetPendingLatched
    OR bHardForceActive OR bHardStrokeActive OR bCollisionLimitActive
    OR bExternalError OR bAxisError OR bSensorInvalid OR (udiFirstFaultId > 0);
bReturnSafeStopRequested := ((eState = CFF_RETURN_LOCAL)
        OR (eState = CFF_RETURN_REFERENCE)
        OR (eState = CFF_EVALUATE)
        OR (eState = CFF_COMPLETE_OK)
        OR (eState = CFF_COMPLETE_NOK))
    AND bSafeExitRequested;

(* Return-capable intent never survives a same-scan real fault or active event. *)
IF (udiFirstFaultId > 0) OR bHardForceActive OR bHardStrokeActive
    OR bCollisionLimitActive OR bExternalError OR bAxisError OR bSensorInvalid THEN
    eExitIntent := CFF_EXIT_FAULT_NO_RETURN;
ELSIF bStopRequestedLatched OR bAbortEvent OR bResetPendingLatched THEN
    eExitIntent := CFF_EXIT_ABORT_NO_RETURN;
END_IF

(* Disable may have selected Abort before a same-scan real fault was normalized. *)
IF (eState = CFF_EXTSETPOINT_DISABLE)
    AND (eNextState = CFF_ABORT)
    AND (eExitIntent = CFF_EXIT_FAULT_NO_RETURN) THEN
    eNextState := CFF_FAULT;
END_IF

(* Abort等待中出现的真实故障必须覆盖Abort，但不改写已锁存的更早首故障。 *)
IF (eState = CFF_ABORT) AND (eExitIntent = CFF_EXIT_FAULT_NO_RETURN) THEN
    eNextState := CFF_FAULT;
END_IF

(* A same-scan hard/error/abort path cannot withdraw the External owner before release. *)
IF bExternalOwnerHold AND bSafeExitRequested THEN
    stMotionIntent.stZCommand.bEnable := TRUE;
    stMotionIntent.stZCommand.eOwnerRequest := Z_OWNER_FORCE_PROCESS;
    stMotionIntent.stZCommand.bUseExternalSetpoint := TRUE;
    stMotionIntent.rExternalTargetVelocity_mm_s := 0.0;
    stMotionIntent.bForceProcessExitComplete := FALSE;
    stMotionIntent.bRAxisProcessRequested := TRUE;
    stCandidateRCommand.bEnable := TRUE;
    stCandidateRCommand.bReset := FALSE;
    stCandidateRCommand.bStop := TRUE;
    stCandidateRCommand.bMoveVelocity := FALSE;
    stCandidateRCommand.rVelocity_rpm := 0.0;
    stCandidateRCommand.rAcceleration_rpm_s := stRAxisProfileSnapshot.fSpeedRampRpmS;
    stCandidateRCommand.rDeceleration_rpm_s := stRAxisProfileSnapshot.fSpeedRampRpmS;
    stMotionIntent.stRCommand := stCandidateRCommand;
    bSafeExitRStopPending := TRUE;
    IF stCandidateRCommand.bEnable <> stLastPublishedRCommand.bEnable
        OR stCandidateRCommand.bReset <> stLastPublishedRCommand.bReset
        OR stCandidateRCommand.bStop <> stLastPublishedRCommand.bStop
        OR stCandidateRCommand.bMoveVelocity <> stLastPublishedRCommand.bMoveVelocity
        OR stCandidateRCommand.rVelocity_rpm <> stLastPublishedRCommand.rVelocity_rpm
        OR stCandidateRCommand.rAcceleration_rpm_s
            <> stLastPublishedRCommand.rAcceleration_rpm_s
        OR stCandidateRCommand.rDeceleration_rpm_s
            <> stLastPublishedRCommand.rDeceleration_rpm_s THEN
        stLastPublishedRCommand := stCandidateRCommand;
        stMotionIntent.stRCommand := stCandidateRCommand;
        udiRCommandId := udiRCommandId + 1;
        IF udiRCommandId = 0 THEN
            udiRCommandId := 1;
        END_IF
    END_IF
    bForceControlEnable := FALSE;
    IF (eExitIntent = CFF_EXIT_ABORT_NO_RETURN)
        AND bUnloadHealthy
        AND (eState >= CFF_CONTACT_SEARCH)
        AND (eState <= CFF_CONTROLLED_FORCE_UNLOAD) THEN
        stMotionIntent.bExternalEnableRequest := TRUE;
        stMotionIntent.bExternalDisableRequest := FALSE;
        bForceControlEnable := TRUE;
        rForceSet_kN := 0.0;
        IF eState < CFF_CONTROLLED_FORCE_UNLOAD THEN
            IF NOT bUnloadTransferInitialized THEN
                rTargetRelativePosition_mm := GVL_Process.stActual.fSRelSensorMm;
                rForceTransferVelocity_mm_s :=
                    GVL_Status.stFast.stZExtSetpoint.rAcceptedVelocity_mm_s;
                bForceProfileTransferPending := TRUE;
                bUnloadTransferInitialized := TRUE;
            END_IF
            eNextState := CFF_CONTROLLED_FORCE_UNLOAD;
        END_IF
    ELSE
        stMotionIntent.bExternalEnableRequest := FALSE;
        stMotionIntent.bExternalDisableRequest := TRUE;
        bForceControlEnable := FALSE;
        eNextState := CFF_EXTSETPOINT_DISABLE;
    END_IF
END_IF

(* If release and a safety cause arrive in the same scan, the state branch may
   already have rebuilt an Enable request.  The strictly positive release gate
   therefore overrides the complete payload with fresh standard stop identities. *)
IF GVL_Status.stFast.stZExtSetpoint.bReleaseOwner THEN
    IF bExternalProcessState
        AND GVL_Status.stFast.stZExtSetpoint.bReleaseOwner
        AND bSafeExitRequested THEN
        udiZCommandId := udiZCommandId + 1;
        IF udiZCommandId = 0 THEN
            udiZCommandId := 1;
        END_IF
        udiRCommandId := udiRCommandId + 1;
        IF udiRCommandId = 0 THEN
            udiRCommandId := 1;
        END_IF
        bApproachFaultStopPending := TRUE;
        stMotionIntent.bExternalEnableRequest := FALSE;
        stMotionIntent.bExternalDisableRequest := FALSE;
        stMotionIntent.rExternalTargetVelocity_mm_s := 0.0;
        stMotionIntent.bForceProcessExitComplete := TRUE;
        stMotionIntent.stZCommand.bEnable := TRUE;
        stMotionIntent.stZCommand.bReset := FALSE;
        stMotionIntent.stZCommand.bStop := TRUE;
        stMotionIntent.stZCommand.bHome := FALSE;
        stMotionIntent.stZCommand.bMoveAbsolute := FALSE;
        stMotionIntent.stZCommand.bMoveVelocity := FALSE;
        stMotionIntent.stZCommand.eOwnerRequest := Z_OWNER_FAULT_STOP;
        stMotionIntent.stZCommand.bUseExternalSetpoint := FALSE;
        stMotionIntent.stZCommand.rHomePosition_mm := 0.0;
        stMotionIntent.stZCommand.rPosition_mm := 0.0;
        stMotionIntent.stZCommand.rVelocity_mm_s := 0.0;
        stMotionIntent.stZCommand.rAcceleration_mm_s2 := stSequenceConfigSnapshot.fStandardMoveAccelerationMmS2;
        stMotionIntent.stZCommand.rDeceleration_mm_s2 := stSequenceConfigSnapshot.fStandardMoveDecelerationMmS2;
        stMotionIntent.bRAxisProcessRequested := TRUE;
        stMotionIntent.stRCommand.bEnable := TRUE;
        stMotionIntent.stRCommand.bReset := FALSE;
        stMotionIntent.stRCommand.bStop := TRUE;
        stMotionIntent.stRCommand.bMoveVelocity := FALSE;
        stMotionIntent.stRCommand.rVelocity_rpm := 0.0;
        stMotionIntent.stRCommand.rAcceleration_rpm_s := stRAxisProfileSnapshot.fSpeedRampRpmS;
        stMotionIntent.stRCommand.rDeceleration_rpm_s := stRAxisProfileSnapshot.fSpeedRampRpmS;
        bForceControlEnable := FALSE;
        IF eExitIntent = CFF_EXIT_ABORT_NO_RETURN THEN
            eNextState := CFF_ABORT;
        ELSE
            eExitIntent := CFF_EXIT_FAULT_NO_RETURN;
            eNextState := CFF_FAULT;
        END_IF
    END_IF
END_IF

(* Return/Evaluate/Complete的同扫安全事件在状态分支之后覆盖Done，并只创建一次FaultStop事务。 *)
IF bReturnSafeStopRequested THEN
    IF NOT bApproachFaultStopPending THEN
        udiZCommandId := udiZCommandId + 1;
        IF udiZCommandId = 0 THEN
            udiZCommandId := 1;
        END_IF
        bApproachFaultStopPending := TRUE;
    END_IF
    stMotionIntent.stZCommand.bEnable := TRUE;
    stMotionIntent.stZCommand.bReset := FALSE;
    stMotionIntent.stZCommand.bStop := TRUE;
    stMotionIntent.stZCommand.bHome := FALSE;
    stMotionIntent.stZCommand.bMoveAbsolute := FALSE;
    stMotionIntent.stZCommand.bMoveVelocity := FALSE;
    stMotionIntent.stZCommand.bUseExternalSetpoint := FALSE;
    stMotionIntent.stZCommand.rHomePosition_mm := 0.0;
    stMotionIntent.stZCommand.rPosition_mm := 0.0;
    stMotionIntent.stZCommand.rVelocity_mm_s := 0.0;
    stMotionIntent.stZCommand.rAcceleration_mm_s2 :=
        stSequenceConfigSnapshot.fStandardMoveAccelerationMmS2;
    stMotionIntent.stZCommand.rDeceleration_mm_s2 :=
        stSequenceConfigSnapshot.fStandardMoveDecelerationMmS2;
    stMotionIntent.stZCommand.eOwnerRequest := Z_OWNER_FAULT_STOP;
    stMotionIntent.bExternalEnableRequest := FALSE;
    stMotionIntent.bExternalDisableRequest := FALSE;
    stMotionIntent.rExternalTargetVelocity_mm_s := 0.0;
    stMotionIntent.bForceProcessExitComplete := TRUE;
    stMotionIntent.bRAxisProcessRequested := TRUE;
    stMotionIntent.stRCommand.bEnable := TRUE;
    stMotionIntent.stRCommand.bReset := FALSE;
    stMotionIntent.stRCommand.bStop := TRUE;
    stMotionIntent.stRCommand.bMoveVelocity := FALSE;
    stMotionIntent.stRCommand.rVelocity_rpm := 0.0;
    stMotionIntent.stRCommand.rAcceleration_rpm_s := stRAxisProfileSnapshot.fSpeedRampRpmS;
    stMotionIntent.stRCommand.rDeceleration_rpm_s := stRAxisProfileSnapshot.fSpeedRampRpmS;
    bForceControlEnable := FALSE;
    IF eExitIntent = CFF_EXIT_FAULT_NO_RETURN THEN
        eNextState := CFF_FAULT;
    ELSE
        eExitIntent := CFF_EXIT_ABORT_NO_RETURN;
        eNextState := CFF_ABORT;
    END_IF
END_IF

(* Precheck owns no motion, so active Stop/Abort/Reset can route directly to a
   terminal wait without depending on the asynchronous Contact Reset ACK. *)
IF eState = CFF_PRECHECK AND bPrecheckExitRequested THEN
    IF eExitIntent = CFF_EXIT_ABORT_NO_RETURN THEN
        eNextState := CFF_ABORT;
    ELSE
        eExitIntent := CFF_EXIT_FAULT_NO_RETURN;
        eNextState := CFF_FAULT;
    END_IF
END_IF

(* Approach has not entered External and may use the standard Fault Stop path. *)
IF eState = CFF_APPROACH AND bSafeExitRequested THEN
    IF NOT bApproachFaultStopPending THEN
        udiZCommandId := udiZCommandId + 1;
        IF udiZCommandId = 0 THEN
            udiZCommandId := 1;
        END_IF
        bApproachFaultStopPending := TRUE;
    END_IF
    stMotionIntent.stZCommand.bEnable := TRUE;
    stMotionIntent.stZCommand.bReset := FALSE;
    stMotionIntent.stZCommand.bStop := TRUE;
    stMotionIntent.stZCommand.bHome := FALSE;
    stMotionIntent.stZCommand.bMoveAbsolute := FALSE;
    stMotionIntent.stZCommand.bMoveVelocity := FALSE;
    stMotionIntent.stZCommand.eOwnerRequest := Z_OWNER_FAULT_STOP;
    stMotionIntent.stZCommand.bUseExternalSetpoint := FALSE;
    stMotionIntent.stZCommand.rHomePosition_mm := 0.0;
    stMotionIntent.stZCommand.rPosition_mm := 0.0;
    stMotionIntent.stZCommand.rVelocity_mm_s := 0.0;
    stMotionIntent.stZCommand.rAcceleration_mm_s2 := stSequenceConfigSnapshot.fStandardMoveAccelerationMmS2;
    stMotionIntent.stZCommand.rDeceleration_mm_s2 := stSequenceConfigSnapshot.fStandardMoveDecelerationMmS2;
    stMotionIntent.bExternalDisableRequest := FALSE;
    IF tonRAxisStop.Q
        OR (udiFirstFaultId = 16#0000A014) THEN
        eExitIntent := CFF_EXIT_FAULT_NO_RETURN;
        eNextState := CFF_FAULT;
    ELSIF tonApproach.Q THEN
        IF udiFirstFaultId = 0 THEN
            udiFirstFaultId := 16#0000A007;
        END_IF
        eExitIntent := CFF_EXIT_FAULT_NO_RETURN;
        eNextState := CFF_FAULT;
    ELSIF (GVL_Status.stFast.udiAcceptedSequenceZCommandId = udiZCommandId)
        AND GVL_Status.stFast.stZAxis.bStandstill
        AND (GVL_Status.stFast.udiAcceptedSequenceRCommandId = udiRCommandId)
        AND GVL_Status.stFast.stRAxis.bStandstill THEN
        bApproachFaultStopPending := FALSE;
        IF eExitIntent = CFF_EXIT_ABORT_NO_RETURN THEN
            eNextState := CFF_ABORT;
        ELSIF eExitIntent = CFF_EXIT_FAULT_NO_RETURN THEN
            eNextState := CFF_FAULT;
        ELSE
            IF udiFirstFaultId = 0 THEN
                udiFirstFaultId := 16#0000A016;
            END_IF
            eExitIntent := CFF_EXIT_FAULT_NO_RETURN;
            eNextState := CFF_FAULT;
        END_IF
    ELSE
        eNextState := eState;
    END_IF
END_IF

IF (eState = CFF_IDLE) AND NOT bSafeTerminalReset
    AND (bStopRequestedLatched OR bAbortEvent OR bResetPendingLatched) THEN
    eExitIntent := CFF_EXIT_ABORT_NO_RETURN;
    eNextState := CFF_ABORT;
END_IF

IF (eState = CFF_IDLE) AND (udiFirstFaultId <> 0) THEN
    bBusy := TRUE;
    eExitIntent := CFF_EXIT_FAULT_NO_RETURN;
    eNextState := CFF_FAULT;
END_IF

(* Contact publisher: five payload fields first and the RequestId last, at one site only. *)
IF bProcessReferencePending THEN
    GVL_Command.stProcessReference.bLatchContactReference :=
        stPendingProcessReferenceCommand.bLatchContactReference;
    GVL_Command.stProcessReference.bUseProvidedContactReference :=
        stPendingProcessReferenceCommand.bUseProvidedContactReference;
    GVL_Command.stProcessReference.rProvidedContactSensorPosition_mm :=
        stPendingProcessReferenceCommand.rProvidedContactSensorPosition_mm;
    GVL_Command.stProcessReference.rProvidedContactAxisPosition_mm :=
        stPendingProcessReferenceCommand.rProvidedContactAxisPosition_mm;
    GVL_Command.stProcessReference.bResetContactReference :=
        stPendingProcessReferenceCommand.bResetContactReference;
    GVL_Command.stProcessReference.udiContactReferenceRequestId :=
        stPendingProcessReferenceCommand.udiContactReferenceRequestId;
END_IF

(* A profile-transfer request is retained until Force is actually enabled. *)
IF bForceProfileTransferPending AND bForceControlEnable THEN
    bForceProfileTransfer := TRUE;
    bForceProfileTransferPending := FALSE;
END_IF

IF bSafeTerminalReset THEN
    bBusy := FALSE;
    bDone := FALSE;
    bError := FALSE;
    bAborted := FALSE;
    bStopRequestedLatched := FALSE;
    bResetPendingLatched := FALSE;
    bCycleNokLatched := FALSE;
    udiFirstFaultId :=0;
    udiActiveStartCommandId := 0;
    bStartSourceSnapshotConsistent := FALSE;
    eExitIntent := CFF_EXIT_NONE;
    eStep := CFF_STEP_NONE;
    eSubPhase := STEP_SUBPHASE_NONE;
    eEndCause := STEP_END_NONE;
    stFastConfigSnapshot.bValid := FALSE;
    bForceControlEnable := FALSE;
    bForceProfileTransfer := FALSE;
    bForceProfileTransferPending := FALSE;
    rForceTransferVelocity_mm_s := 0.0;
    rForceSet_kN := 0.0;
    rForceRamp_kN_s := 0.0;
    rSpeedSet_rpm := 0.0;
    rTargetRelativePosition_mm := 0.0;
    rHardMaximumRelativePosition_mm := 0.0;
    rRequiredRelativePosition_mm := 0.0;
    rStepBoundary_mm := 0.0;
    rCycleStartZPosition_mm := 0.0;
    rStepTime_s := 0.0;
    rQualifiedForceHoldTime_s := 0.0;
    uliCycleDelta_us := 0;
    uliStepElapsed_us := 0;
    uliStepMaximum_us := 0;
    uliQualifiedHold_us := 0;
    uliQualifiedHoldTarget_us := 0;
    bRpmStopped := FALSE;
    bForceInBand := FALSE;
    bStepResultPublishRequested := FALSE;
    bStepResultNok := FALSE;
    nStepResultIndex := 1;
    bEvaluateNok := FALSE;
    bEvaluateFault := FALSE;
    bStepResultHole := FALSE;
    bMissingStepResult := FALSE;
    nWrittenStepPrefix := 0;
    bHardForceActive := FALSE;
    bHardStrokeActive := FALSE;
    bCollisionLimitActive := FALSE;
    bProcessReferencePending := FALSE;
    bProcessReferenceResetPending := FALSE;
    bProcessReferenceLatchPending := FALSE;
    bApproachFaultStopPending := FALSE;
    bUnknownExternalRStopPending := FALSE;
    bSafeExitRStopPending := FALSE;
    bTerminalFaultStopRequired := FALSE;
    bUnloadTransferInitialized := FALSE;
    bContactResetPulse := TRUE;
    bForceDeclineResetPulse := TRUE;
    bStepCriterionResetPulse := TRUE;
    eNextState := CFF_IDLE;
END_IF

(* Stop is the final diagnostic end cause until Start or safe Reset clears it. *)
IF bStopRequestedLatched THEN
    eEndCause := STEP_END_STOP_REQUEST;
END_IF

(* A transition scan never publishes the completed truth table of its source state. *)
IF (eState <> eNextState)
    AND ((eNextState = CFF_ABORT) OR (eNextState = CFF_FAULT)) THEN
    bBusy := TRUE;
    bDone := FALSE;
    bError := FALSE;
    bAborted := FALSE;
END_IF

